(* IEC 61131-3 sources: std_i2980_v2.06_cp053/Source/IMM/ieccontrol/CentralCoordination1, 6 files *)

(* ---- ABActiveMovements.pu ---- *)
(*
@h    ! WARNING !
@h    The Kemro K2 system (including software) only meets category B according to EN 954-1,
@h    thus it is not intended for usage in safety-relevant control applications in the field
@h    of personal safety (e.g. emergency stop).
@h    To implement potentially necessary safety-relevant control tasks, always use additional
@h    external safety devices that are intended for the particular purpose, and meet the necessary
@h    functional safety.
@h    For further information see EN 954-1 (EN ISO 13849-1) and/or the K2-x00 user manual, chapter
@h    "CE conformity, directives and standards".

*)

IMPORT_OVER_LISTFILE
 SET_ALARM
, cCompNone
, cMoveNone
, cCompInjection
, cMinMoveIdent
, cMaxActiveMovements
, cMoveFwd
, tevMovementState
, tyMovementRegisterList
, tsActiveMovements
, tsStartedMoveData
, tyNumberOfDevices
, tyInjectHoldNumbers
, tevStartedStopped
, tevMovementStateData
, FBGetMoveNumber
, tevStartedStoppedData

END_IMPORT

ALGORITHM_BLOCK ABActiveMovements #DUMMY_EDIT_BLOCK

SYSTEM_VAR
 sv_MovementsAvailable : tyMovementRegisterList;
 sv_iMovementsAvailable : DINT;
 sv_ActiveMovements : tsActiveMovements;
 sv_StartedMovements : tsStartedMoveData;
 sv_bInitDone : BOOL;
 sv_NumberOfDevices : tyNumberOfDevices;
END_VAR

SYSTEM_OBJECT
 EV_Task_3 : TASK;
 evMovementState : tevMovementState;
 PU_Task_13 : TASK;
 evStartedStopped : tevStartedStopped;
 erMaxStartedMovementsExceeded : ALARM;
 erMaxActiveMovementsExceeded : ALARM;
END_OBJECT

VAR
 InjectHoldNumbers : tyInjectHoldNumbers;
END_VAR

(*
Manage a list of active movements for displaying
the active movement on the HMI.
Reacts to evMovementState events
*)

EVENT_ALGORITHM evaMovementState ON EV_Task_3 WITH evMovementState

VAR_INPUT
 evMovementStateData : tevMovementStateData;
END_VAR

VAR_TEMP
 i : DINT;
 k : DINT;
END_VAR

VAR
 iMoveNumber : DINT;
 MovementStateData : tevMovementStateData;
 fbGetMoveNumber : FBGetMoveNumber;
END_VAR
#BEGIN_EDIT_BLOCK
(**************************************** WARNING ********************************************
 *** The KEBA Kemro K2 System including software is not intended for safety control tasks! ***
 ***                       For further information see Comment tab!                        ***
 *********************************************************************************************)

MovementStateData := evMovementStateData;

IF MovementStateData.State = nInactive AND MovementStateData.DeviceId.CompId = cCompInjection AND
   MovementStateData.MoveDir = cMoveFwd AND MovementStateData.MoveId = cMoveInject THEN
   //inject movement was stopped -> check if holding was active
    IF InjectHoldNumbers[MovementStateData.DeviceId.IndexId].bHoldActive THEN
        //holding was active
        iMoveNumber := InjectHoldNumbers[MovementStateData.DeviceId.IndexId].iHoldMovement;
    ELSE
        //holding was not active
        iMoveNumber := InjectHoldNumbers[MovementStateData.DeviceId.IndexId].iInjectMovement;
    END_IF;
    InjectHoldNumbers[MovementStateData.DeviceId.IndexId].bHoldActive := FALSE;
ELSE
    // -> get movement number
    fbGetMoveNumber(DeviceId := MovementStateData.DeviceId,
                    MoveId := MovementStateData.MoveId,
                    MoveDir := MovementStateData.MoveDir,
                    iMoveNumber => iMoveNumber);
END_IF;

IF (iMoveNumber = 0) THEN
    //no movement found
    RETURN;
END_IF;

IF MovementStateData.State = nActive THEN
    IF MovementStateData.MoveId = cMoveHold THEN
        // hold phase active -> search inject movement and change number to hold movement
        FOR i := 1 TO sv_ActiveMovements.iNumberOfActiveMovements DO
            IF sv_ActiveMovements.ActiveMovements[i] = InjectHoldNumbers[MovementStateData.DeviceId.IndexId].iInjectMovement THEN
                sv_ActiveMovements.ActiveMovements[i] := InjectHoldNumbers[MovementStateData.DeviceId.IndexId].iHoldMovement;
                InjectHoldNumbers[MovementStateData.DeviceId.IndexId].bHoldActive := TRUE;
                EXIT;
            END_IF;
        END_FOR;
    ELSE
        IF sv_ActiveMovements.iNumberOfActiveMovements < cMaxActiveMovements THEN
            //movement was started -> add movement to list
            sv_ActiveMovements.ActiveMovements[(sv_ActiveMovements.iNumberOfActiveMovements+1)] := iMoveNumber;
            sv_ActiveMovements.iNumberOfActiveMovements := sv_ActiveMovements.iNumberOfActiveMovements + 1;
        ELSE
            //too many movements active
            SET_ALARM(Name := erMaxActiveMovementsExceeded,
                      SubID1 := cMaxActiveMovements);
        END_IF;
    END_IF;
ELSE
    //movement was stopped -> find movement and delete it from array
    FOR i := 1 TO sv_ActiveMovements.iNumberOfActiveMovements DO
        IF sv_ActiveMovements.ActiveMovements[i] = iMoveNumber THEN
            sv_ActiveMovements.ActiveMovements[i] := 0;
            //move all other movements so that there is no empty field in the list
            FOR k:= (i+1) TO cMaxActiveMovements DO
                sv_ActiveMovements.ActiveMovements[(k-1)] := sv_ActiveMovements.ActiveMovements[k];
                sv_ActiveMovements.ActiveMovements[k] := 0;
            END_FOR;
            sv_ActiveMovements.iNumberOfActiveMovements := sv_ActiveMovements.iNumberOfActiveMovements -1;
            EXIT;
        END_IF;
    END_FOR;

END_IF;

;#END_EDIT_BLOCK END_ALGORITHM

(*
Manage list and count of currently started movments
in sv_StartedMovements when receiving evStartedStopped events
*)

EVENT_ALGORITHM evaStartedStopped ON EV_Task_3 WITH evStartedStopped

VAR_INPUT
 evStartedStoppedData : tevStartedStoppedData;
END_VAR

VAR_TEMP
 i : DINT;
END_VAR

VAR
 dummy : DINT;
END_VAR
#BEGIN_EDIT_BLOCK
(**************************************** WARNING ********************************************
 *** The KEBA Kemro K2 System including software is not intended for safety control tasks! ***
 ***                       For further information see Comment tab!                        ***
 *********************************************************************************************)

IF evStartedStoppedData.State = nStarted THEN
    //movement started
    IF sv_StartedMovements.iStartedMovements < cMaxActiveMovements THEN
        //add movement to sv_StartedMovements
        sv_StartedMovements.iStartedMovements := sv_StartedMovements.iStartedMovements +1;
        sv_StartedMovements.MoveData[sv_StartedMovements.iStartedMovements].DeviceId := evStartedStoppedData.DeviceId;
        sv_StartedMovements.MoveData[sv_StartedMovements.iStartedMovements].MoveDir := evStartedStoppedData.MoveDir;
        sv_StartedMovements.MoveData[sv_StartedMovements.iStartedMovements].MoveId := evStartedStoppedData.MoveId;
    ELSE
        //too many movements started
        //show some information about the movement to make debugging easier
        dummy := Print('set alarm erMaxStartedMovementsExceeded in ABActiveMovements.pu');
        dummy := Print('max. active movements: %d', cMaxActiveMovements);
        dummy := Print('tried to start    %d.%d %d/%d',
                       evStartedStoppedData.DeviceId.CompId, evStartedStoppedData.DeviceId.IndexId,
                       evStartedStoppedData.MoveId, evStartedStoppedData.MoveDir);
        FOR i := 1 TO cMaxActiveMovements DO
            dummy := Print('already started %d %d.%d %d/%d',
                           i, sv_StartedMovements.MoveData[i].DeviceId.CompId, sv_StartedMovements.MoveData[i].DeviceId.IndexId,
                           sv_StartedMovements.MoveData[i].MoveId, sv_StartedMovements.MoveData[i].MoveDir);
        END_FOR;

        //set alarm after tracing out
        SET_ALARM(Name := erMaxStartedMovementsExceeded,
                  SubID1 := cMaxActiveMovements);
    END_IF;
ELSE
    //movement stopped
    //remove movement from list with started movements
    FOR i := 1 TO sv_StartedMovements.iStartedMovements DO
        IF sv_StartedMovements.MoveData[i].DeviceId = evStartedStoppedData.DeviceId AND
           sv_StartedMovements.MoveData[i].MoveDir = evStartedStoppedData.MoveDir AND
           sv_StartedMovements.MoveData[i].MoveId = evStartedStoppedData.MoveId THEN
            sv_StartedMovements.MoveData[i].DeviceId.CompId := cCompNone;
            sv_StartedMovements.MoveData[i].DeviceId.IndexId := 1;
            sv_StartedMovements.MoveData[i].MoveDir := cMoveNone;
            sv_StartedMovements.MoveData[i].MoveId := cMinMoveIdent;
            //copy last entry in the list to this empty field
            sv_StartedMovements.MoveData[i] := sv_StartedMovements.MoveData[sv_StartedMovements.iStartedMovements];
            sv_StartedMovements.iStartedMovements := sv_StartedMovements.iStartedMovements -1;
            EXIT;
        END_IF;
    END_FOR;
END_IF;

;#END_EDIT_BLOCK END_ALGORITHM

POSTUPDATE_ALGORITHM pGetInjectHoldNumbers ON PU_Task_13 WITH sv_bInitDone

VAR_TEMP
 i : DINT;
 iDevice : DINT;
END_VAR
#BEGIN_EDIT_BLOCK
(**************************************** WARNING ********************************************
 *** The KEBA Kemro K2 System including software is not intended for safety control tasks! ***
 ***                       For further information see Comment tab!                        ***
 *********************************************************************************************)

//get icon pathes for inject and hold of all registered injection function units
FOR iDevice := 1 TO sv_NumberOfDevices[cCompInjection] DO

    FOR i := 1 TO sv_iMovementsAvailable DO
        IF sv_MovementsAvailable[i].DeviceId.CompId = cCompInjection AND
           sv_MovementsAvailable[i].pMovementData^.MoveId = cMoveInject THEN
            //save number of inject movement
            InjectHoldNumbers[sv_MovementsAvailable[i].DeviceId.IndexId].iInjectMovement := i;
        END_IF;
        IF sv_MovementsAvailable[i].DeviceId.CompId = cCompInjection AND
           sv_MovementsAvailable[i].pMovementData^.MoveId = cMoveHold THEN
            //save number of holding movement
            InjectHoldNumbers[sv_MovementsAvailable[i].DeviceId.IndexId].iHoldMovement := i;
        END_IF;
    END_FOR;

END_FOR;

;#END_EDIT_BLOCK END_ALGORITHM

END_ALGORITHM_BLOCK

#END_OF_IEC_PART

@Puma @IecEditor 6 86 @Pou 25
@@@BEG_Comment@@@
@h    ! WARNING !
@h    The Kemro K2 system (including software) only meets category B according to EN 954-1,
@h    thus it is not intended for usage in safety-relevant control applications in the field
@h    of personal safety (e.g. emergency stop).
@h    To implement potentially necessary safety-relevant control tasks, always use additional
@h    external safety devices that are intended for the particular purpose, and meet the necessary
@h    functional safety.
@h    For further information see EN 954-1 (EN ISO 13849-1) and/or the K2-x00 user manual, chapter
@h    "CE conformity, directives and standards".

@@@END_Comment@@@

@BEG_Contents

@BEG_Func
@RT(17)FuncTreeContainer
1
@Var @RT(9)SET_ALARM @RT(0) @T @T @DERIVED 0 @F @RT(23)KEBA_STANDARD_PROCEDURE @F
@T
@BEG_Attrib
0 @RT(0) @RT(0)
@END_Attrib
1 1 @F @F @F @F

@END_Func

@BEG_Const
@RT(18)ConstTreeContainer
6
@Var @RT(9)cCompNone @RT(0) @T @F @DT @RT(4)DINT @RT(0) @T @T @BASIC 0 @F
@F @F
@T
@BEG_Attrib
0 @RT(10)cMinCompId @RT(4)None
@END_Attrib
1 1 @F @F @F @F

@Var @RT(9)cMoveNone @RT(0) @T @F @DT @RT(4)DINT @RT(0) @T @T @BASIC 0 @F
@F @F
@T
@BEG_Attrib
0 @RT(13)cMinMoveIdent @RT(4)None
@END_Attrib
1 1 @F @F @F @F

@Var @RT(14)cCompInjection @RT(0) @T @F @DT @RT(4)DINT @RT(0) @T @T @BASIC 0 @F
@F @F
@T
@BEG_Attrib
0 @RT(3)104 @RT(19)Component Injection
@END_Attrib
1 1 @F @F @F @F

@Var @RT(13)cMinMoveIdent @RT(0) @T @F @DT @RT(4)DINT @RT(0) @T @T @BASIC 0 @F
@F @F
@T
@BEG_Attrib
0 @RT(1)1 @RT(32)lower limit for MoveId / MoveDir
@END_Attrib
1 1 @F @F @F @F

@Var @RT(19)cMaxActiveMovements @RT(0) @T @F @DT @RT(4)DINT @RT(0) @T @T @BASIC 0 @F
@F @F
@T
@BEG_Attrib
0 @RT(1)6 @RT(52)number of movements that are active at the same time
@END_Attrib
1 1 @F @F @F @F

@Var @RT(8)cMoveFwd @RT(0) @T @F @DT @RT(4)DINT @RT(0) @T @T @BASIC 0 @F
@F @F
@T
@BEG_Attrib
0 @RT(2)12 @RT(16)movement forward
@END_Attrib
1 1 @F @F @F @F

@END_Const

@BEG_Export

@BEG_Kind
@ALGORITHM_BLOCK @RT(17)ABActiveMovements @STRUCTURED_TEXT
@RT(0) @RT(0) @RT(0)
@END_Kind

@BEG_Dcl
@RT(16)DclTreeContainer
13
@Var @RT(9)EV_Task_3 @RT(0) @T @T @RENAMED 0 @T @T @DT @RT(4)TASK @RT(0) @T @T @BASIC 0 @F
@F @F
@T
@BEG_Attrib
3 @RT(0) @RT(0) @RT(0)
@END_Attrib
1 7 @F @F @F @F

@Var @RT(15)evMovementState @RT(0) @T @T @DERIVED 0 @T @T @DT @RT(16)tevMovementState @RT(0) @T @T @UNKNOWN 0 @F
@F @F
@T
@BEG_Attrib
3 @RT(0) @RT(0) @RT(0)
@END_Attrib
1 7 @F @F @F @F

@Var @RT(21)sv_MovementsAvailable @RT(0) @T @T @DERIVED 0 @T @T @DT @RT(22)tyMovementRegisterList @RT(0) @T @T @UNKNOWN 0 @F
@F @F
@T
@BEG_Attrib
3 @RT(0) @RT(0) @RT(0)
@END_Attrib
1 8 @F @F @F @F

@Var @RT(22)sv_iMovementsAvailable @RT(0) @T @F @DT @RT(4)DINT @RT(0) @T @T @BASIC 0 @F
@F @F
@T
@BEG_Attrib
3 @RT(0) @RT(0) @RT(0)
@END_Attrib
1 8 @F @F @F @F

@Var @RT(18)sv_ActiveMovements @RT(0) @T @T @DERIVED 0 @T @T @DT @RT(17)tsActiveMovements @RT(0) @T @T @UNKNOWN 0 @F
@F @F
@T
@BEG_Attrib
3 @RT(0) @RT(0) @RT(0)
@END_Attrib
1 8 @F @F @F @F

@Var @RT(19)sv_StartedMovements @RT(0) @T @T @DERIVED 0 @T @T @DT @RT(17)tsStartedMoveData @RT(0) @T @T @UNKNOWN 0 @F
@F @F
@T
@BEG_Attrib
3 @RT(0) @RT(0) @RT(0)
@END_Attrib
1 8 @F @F @F @F

@Var @RT(10)PU_Task_13 @RT(0) @T @T @RENAMED 0 @T @T @DT @RT(4)TASK @RT(0) @T @T @BASIC 0 @F
@F @F
@T
@BEG_Attrib
3 @RT(0) @RT(0) @RT(0)
@END_Attrib
1 7 @F @F @F @F

@Var @RT(12)sv_bInitDone @RT(0) @T @T @RENAMED 0 @T @T @DT @RT(4)BOOL @RT(0) @T @T @BASIC 0 @F
@F @F
@T
@BEG_Attrib
3 @RT(0) @RT(0) @RT(0)
@END_Attrib
1 8 @F @F @F @F

@Var @RT(18)sv_NumberOfDevices @RT(0) @T @T @DERIVED 0 @T @T @DT @RT(17)tyNumberOfDevices @RT(0) @T @T @UNKNOWN 0 @F
@F @F
@T
@BEG_Attrib
3 @RT(0) @RT(0) @RT(0)
@END_Attrib
1 8 @F @F @F @F

@Var @RT(17)InjectHoldNumbers @RT(0) @T @T @DERIVED 0 @T @T @DT @RT(19)tyInjectHoldNumbers @RT(0) @T @T @UNKNOWN 0 @F
@F @F
@T
@BEG_Attrib
3 @RT(0) @RT(0) @RT(0)
@END_Attrib
1 0 @F @F @F @F

@Var @RT(16)evStartedStopped @RT(0) @T @T @RENAMED 0 @T @T @DT @RT(17)tevStartedStopped @RT(0) @T @T @UNKNOWN 0 @F
@F @F
@T
@BEG_Attrib
3 @RT(0) @RT(0) @RT(0)
@END_Attrib
1 7 @F @F @F @F

@Var @RT(29)erMaxStartedMovementsExceeded @RT(0) @T @T @RENAMED 0 @T @T @DT @RT(5)ALARM @RT(0) @T @T @BASIC 0 @F
@F @F
@T
@BEG_Attrib
3 @RT(0) @RT(0) @RT(0)
@END_Attrib
1 7 @F @F @F @F

@Var @RT(28)erMaxActiveMovementsExceeded @RT(0) @T @T @RENAMED 0 @T @T @DT @RT(5)ALARM @RT(0) @T @T @BASIC 0 @F
@F @F
@T
@BEG_Attrib
3 @RT(0) @RT(0) @RT(0)
@END_Attrib
1 7 @F @F @F @F

@END_Dcl

@END_Export

@BEG_Body

3

@BEG_Export

@BEG_Algo
@EVENT_ALGORITHM @RT(16)evaMovementState @STRUCTURED_TEXT
@RT(0) @RT(15)evMovementState @RT(9)EV_Task_3 @F @F
@END_Algo

@BEG_Dcl
@RT(16)DclTreeContainer
6
@Var @RT(19)evMovementStateData @RT(0) @T @T @DERIVED 0 @T @T @DT @RT(20)tevMovementStateData @RT(0) @T @T @UNKNOWN 0 @F
@F @F
@T
@BEG_Attrib
3 @RT(0) @RT(0) @RT(0)
@END_Attrib
1 1 @F @F @F @F

@Var @RT(1)i @RT(0) @T @F @DT @RT(4)DINT @RT(0) @T @T @BASIC 0 @F
@F @F
@T
@BEG_Attrib
3 @RT(0) @RT(0) @RT(0)
@END_Attrib
1 4 @F @F @F @F

@Var @RT(1)k @RT(0) @T @F @DT @RT(4)DINT @RT(0) @T @T @BASIC 0 @F
@F @F
@T
@BEG_Attrib
3 @RT(0) @RT(0) @RT(0)
@END_Attrib
1 4 @F @F @F @F

@Var @RT(11)iMoveNumber @RT(0) @T @F @DT @RT(4)DINT @RT(0) @T @T @BASIC 0 @F
@F @F
@T
@BEG_Attrib
3 @RT(0) @RT(0) @RT(0)
@END_Attrib
1 0 @F @F @F @F

@Var @RT(17)MovementStateData @RT(0) @T @T @DERIVED 0 @T @T @DT @RT(20)tevMovementStateData @RT(0) @T @T @UNKNOWN 0 @F
@F @F
@T
@BEG_Attrib
3 @RT(0) @RT(0) @RT(0)
@END_Attrib
1 0 @F @F @F @F

@Var @RT(15)fbGetMoveNumber @RT(0) @T @T @DERIVED 0 @T @T @DT @RT(15)FBGetMoveNumber @RT(0) @T @T @UNKNOWN 0 @F
@F @F
@T
@BEG_Attrib
3 @RT(0) @RT(0) @RT(0)
@END_Attrib
1 0 @F @F @F @F

@END_Dcl

@END_Export

@BEG_Export

@BEG_Algo
@EVENT_ALGORITHM @RT(17)evaStartedStopped @STRUCTURED_TEXT
@RT(0) @RT(16)evStartedStopped @RT(9)EV_Task_3 @F @F
@END_Algo

@BEG_Dcl
@RT(16)DclTreeContainer
3
@Var @RT(20)evStartedStoppedData @RT(0) @T @T @DERIVED 0 @T @T @DT @RT(21)tevStartedStoppedData @RT(0) @T @T @UNKNOWN 0 @F
@F @F
@T
@BEG_Attrib
3 @RT(0) @RT(0) @RT(0)
@END_Attrib
1 1 @F @F @F @F

@Var @RT(1)i @RT(0) @T @F @DT @RT(4)DINT @RT(0) @T @T @BASIC 0 @F
@F @F
@T
@BEG_Attrib
3 @RT(0) @RT(0) @RT(0)
@END_Attrib
1 4 @F @F @F @F

@Var @RT(5)dummy @RT(0) @T @F @DT @RT(4)DINT @RT(0) @T @T @BASIC 0 @F
@F @F
@T
@BEG_Attrib
3 @RT(0) @RT(0) @RT(0)
@END_Attrib
1 0 @F @F @F @F

@END_Dcl

@END_Export

@BEG_Export

@BEG_Algo
@POSTUPDATE_ALGORITHM @RT(21)pGetInjectHoldNumbers @STRUCTURED_TEXT
@RT(0) @RT(12)sv_bInitDone @RT(10)PU_Task_13 @F @F
@END_Algo

@BEG_Dcl
@RT(16)DclTreeContainer
2
@Var @RT(1)i @RT(0) @T @F @DT @RT(4)DINT @RT(0) @T @T @BASIC 0 @F
@F @F
@T
@BEG_Attrib
3 @RT(0) @RT(0) @RT(0)
@END_Attrib
1 4 @F @F @F @F

@Var @RT(7)iDevice @RT(0) @T @F @DT @RT(4)DINT @RT(0) @T @T @BASIC 0 @F
@F @F
@T
@BEG_Attrib
3 @RT(0) @RT(0) @RT(0)
@END_Attrib
1 4 @F @F @F @F

@END_Dcl

@END_Export

@BEG_Body
@TL(72)
(**************************************** WARNING ********************************************
 *** The KEBA Kemro K2 System including software is not intended for safety control tasks! ***
 ***                       For further information see Comment tab!                        ***
 *********************************************************************************************)

MovementStateData := evMovementStateData;

IF MovementStateData.State = nInactive AND MovementStateData.DeviceId.CompId = cCompInjection AND
   MovementStateData.MoveDir = cMoveFwd AND MovementStateData.MoveId = cMoveInject THEN
   //inject movement was stopped -> check if holding was active
    IF InjectHoldNumbers[MovementStateData.DeviceId.IndexId].bHoldActive THEN
        //holding was active
        iMoveNumber := InjectHoldNumbers[MovementStateData.DeviceId.IndexId].iHoldMovement;
    ELSE
        //holding was not active
        iMoveNumber := InjectHoldNumbers[MovementStateData.DeviceId.IndexId].iInjectMovement;
    END_IF;
    InjectHoldNumbers[MovementStateData.DeviceId.IndexId].bHoldActive := FALSE;
ELSE
    // -> get movement number
    fbGetMoveNumber(DeviceId := MovementStateData.DeviceId,
                    MoveId := MovementStateData.MoveId,
                    MoveDir := MovementStateData.MoveDir,
                    iMoveNumber => iMoveNumber);
END_IF;

IF (iMoveNumber = 0) THEN
    //no movement found
    RETURN;
END_IF;

IF MovementStateData.State = nActive THEN
    IF MovementStateData.MoveId = cMoveHold THEN
        // hold phase active -> search inject movement and change number to hold movement
        FOR i := 1 TO sv_ActiveMovements.iNumberOfActiveMovements DO
            IF sv_ActiveMovements.ActiveMovements[i] = InjectHoldNumbers[MovementStateData.DeviceId.IndexId].iInjectMovement THEN
                sv_ActiveMovements.ActiveMovements[i] := InjectHoldNumbers[MovementStateData.DeviceId.IndexId].iHoldMovement;
                InjectHoldNumbers[MovementStateData.DeviceId.IndexId].bHoldActive := TRUE;
                EXIT;
            END_IF;
        END_FOR;
    ELSE
        IF sv_ActiveMovements.iNumberOfActiveMovements < cMaxActiveMovements THEN
            //movement was started -> add movement to list
            sv_ActiveMovements.ActiveMovements[(sv_ActiveMovements.iNumberOfActiveMovements+1)] := iMoveNumber;
            sv_ActiveMovements.iNumberOfActiveMovements := sv_ActiveMovements.iNumberOfActiveMovements + 1;
        ELSE
            //too many movements active
            SET_ALARM(Name := erMaxActiveMovementsExceeded,
                      SubID1 := cMaxActiveMovements);
        END_IF;
    END_IF;
ELSE
    //movement was stopped -> find movement and delete it from array
    FOR i := 1 TO sv_ActiveMovements.iNumberOfActiveMovements DO
        IF sv_ActiveMovements.ActiveMovements[i] = iMoveNumber THEN
            sv_ActiveMovements.ActiveMovements[i] := 0;
            //move all other movements so that there is no empty field in the list
            FOR k:= (i+1) TO cMaxActiveMovements DO
                sv_ActiveMovements.ActiveMovements[(k-1)] := sv_ActiveMovements.ActiveMovements[k];
                sv_ActiveMovements.ActiveMovements[k] := 0;
            END_FOR;
            sv_ActiveMovements.iNumberOfActiveMovements := sv_ActiveMovements.iNumberOfActiveMovements -1;
            EXIT;
        END_IF;
    END_FOR;

END_IF;

@END_Body

@@@BEG_Comment@@@
@TL(3)
Manage a list of active movements for displaying
the active movement on the HMI.
Reacts to evMovementState events
@@@END_Comment@@@

@BEG_Body
@TL(54)
(**************************************** WARNING ********************************************
 *** The KEBA Kemro K2 System including software is not intended for safety control tasks! ***
 ***                       For further information see Comment tab!                        ***
 *********************************************************************************************)

IF evStartedStoppedData.State = nStarted THEN
    //movement started
    IF sv_StartedMovements.iStartedMovements < cMaxActiveMovements THEN
        //add movement to sv_StartedMovements
        sv_StartedMovements.iStartedMovements := sv_StartedMovements.iStartedMovements +1;
        sv_StartedMovements.MoveData[sv_StartedMovements.iStartedMovements].DeviceId := evStartedStoppedData.DeviceId;
        sv_StartedMovements.MoveData[sv_StartedMovements.iStartedMovements].MoveDir := evStartedStoppedData.MoveDir;
        sv_StartedMovements.MoveData[sv_StartedMovements.iStartedMovements].MoveId := evStartedStoppedData.MoveId;
    ELSE
        //too many movements started
        //show some information about the movement to make debugging easier
        dummy := Print('set alarm erMaxStartedMovementsExceeded in ABActiveMovements.pu');
        dummy := Print('max. active movements: %d', cMaxActiveMovements);
        dummy := Print('tried to start    %d.%d %d/%d',
                       evStartedStoppedData.DeviceId.CompId, evStartedStoppedData.DeviceId.IndexId,
                       evStartedStoppedData.MoveId, evStartedStoppedData.MoveDir);
        FOR i := 1 TO cMaxActiveMovements DO
            dummy := Print('already started %d %d.%d %d/%d',
                           i, sv_StartedMovements.MoveData[i].DeviceId.CompId, sv_StartedMovements.MoveData[i].DeviceId.IndexId,
                           sv_StartedMovements.MoveData[i].MoveId, sv_StartedMovements.MoveData[i].MoveDir);
        END_FOR;

        //set alarm after tracing out
        SET_ALARM(Name := erMaxStartedMovementsExceeded,
                  SubID1 := cMaxActiveMovements);
    END_IF;
ELSE
    //movement stopped
    //remove movement from list with started movements
    FOR i := 1 TO sv_StartedMovements.iStartedMovements DO
        IF sv_StartedMovements.MoveData[i].DeviceId = evStartedStoppedData.DeviceId AND
           sv_StartedMovements.MoveData[i].MoveDir = evStartedStoppedData.MoveDir AND
           sv_StartedMovements.MoveData[i].MoveId = evStartedStoppedData.MoveId THEN
            sv_StartedMovements.MoveData[i].DeviceId.CompId := cCompNone;
            sv_StartedMovements.MoveData[i].DeviceId.IndexId := 1;
            sv_StartedMovements.MoveData[i].MoveDir := cMoveNone;
            sv_StartedMovements.MoveData[i].MoveId := cMinMoveIdent;
            //copy last entry in the list to this empty field
            sv_StartedMovements.MoveData[i] := sv_StartedMovements.MoveData[sv_StartedMovements.iStartedMovements];
            sv_StartedMovements.iStartedMovements := sv_StartedMovements.iStartedMovements -1;
            EXIT;
        END_IF;
    END_FOR;
END_IF;

@END_Body

@@@BEG_Comment@@@
@TL(2)
Manage list and count of currently started movments
in sv_StartedMovements when receiving evStartedStopped events
@@@END_Comment@@@

@BEG_Body
@TL(23)
(**************************************** WARNING ********************************************
 *** The KEBA Kemro K2 System including software is not intended for safety control tasks! ***
 ***                       For further information see Comment tab!                        ***
 *********************************************************************************************)

//get icon pathes for inject and hold of all registered injection function units
FOR iDevice := 1 TO sv_NumberOfDevices[cCompInjection] DO

    FOR i := 1 TO sv_iMovementsAvailable DO
        IF sv_MovementsAvailable[i].DeviceId.CompId = cCompInjection AND
           sv_MovementsAvailable[i].pMovementData^.MoveId = cMoveInject THEN
            //save number of inject movement
            InjectHoldNumbers[sv_MovementsAvailable[i].DeviceId.IndexId].iInjectMovement := i;
        END_IF;
        IF sv_MovementsAvailable[i].DeviceId.CompId = cCompInjection AND
           sv_MovementsAvailable[i].pMovementData^.MoveId = cMoveHold THEN
            //save number of holding movement
            InjectHoldNumbers[sv_MovementsAvailable[i].DeviceId.IndexId].iHoldMovement := i;
        END_IF;
    END_FOR;

END_FOR;

@END_Body

@@@BEG_Comment@@@
@TL(0)

@@@END_Comment@@@
@END_Body

@END_Contents
@@@BEG_Password@@@
M2hzZmhrMw==
@@@END_Password@@@

(* ---- ABAvailableDevices.pu ---- *)
(*
@h    ! WARNING !
@h    The Kemro K2 system (including software) only meets category B according to EN 954-1,
@h    thus it is not intended for usage in safety-relevant control applications in the field
@h    of personal safety (e.g. emergency stop).
@h    To implement potentially necessary safety-relevant control tasks, always use additional
@h    external safety devices that are intended for the particular purpose, and meet the necessary
@h    functional safety.
@h    For further information see EN 954-1 (EN ISO 13849-1) and/or the K2-x00 user manual, chapter
@h    "CE conformity, directives and standards".

This AB listens to the device register events and sets
the sv_CoreData[X].bAvailable - flag if a core is available (registered).
Additionally it listens to evCoreTypeChanged events and sets
sv_bCoresActive if any registered core is switched on.
After a failed creation of a new sequence (by using program switches), The core priorities are
checked. If there are some equal priorities, an according alarm is displayed
*)

IMPORT_OVER_LISTFILE
 SET_ALARM
, cCompAirValve
, cMaxDeviceIndex
, cMoveIn
, tyCoreData
, tevDeviceRegister
, tevCoreTypeChanged
, tyDeviceAvailable
, tyNumberOfDevices
, KSYS_Status
, tevDeviceRegisterData
, tevCoreTypeChangedData

END_IMPORT

ALGORITHM_BLOCK ABAvailableDevices #DUMMY_EDIT_BLOCK

SYSTEM_VAR
 sv_CoreData : tyCoreData;
 sv_CoreOff : tyDeviceAvailable;
 sv_bCoresActive : BOOL (* TRUE: any core is switched on *);
 sv_bInitStart : BOOL;
 sv_bUseProgramSwitches : BOOL;
 sv_bCoresParallelToMold : BOOL;
 sv_bDeviceRegisterDone : BOOL;
 sv_NumberOfDevices : tyNumberOfDevices;
END_VAR

SYSTEM_OBJECT
 EV_Task_3 : TASK;
 evDeviceRegister : tevDeviceRegister;
 EV_Task_7 : TASK;
 evCoreTypeChanged : tevCoreTypeChanged;
 PU_Task_7 : TASK;
 TaskMid : TASK;
 erEqualCorePriority : ALARM;
 PU_Task_3 : TASK;
END_OBJECT

VAR
 mpiODCSequenceUpdated : REFTO DINT;
 mpiODCInitOk : REFTO DINT;
END_VAR

POSTUPDATE_ALGORITHM pInitStart ON PU_Task_7 WITH sv_bInitStart

VAR
 state : KSYS_Status;
END_VAR
#BEGIN_EDIT_BLOCK
(**************************************** WARNING ********************************************
 *** The KEBA Kemro K2 System including software is not intended for safety control tasks! ***
 ***                       For further information see Comment tab!                        ***
 *********************************************************************************************)

//get references
mpiODCSequenceUpdated := GET_SYNC_REFTO('ODC1.sv_iODCSequenceUpdated', T#0s, state);
mpiODCInitOk := GET_SYNC_REFTO('ODC1.sv_iInitOK', T#0s, state);

;#END_EDIT_BLOCK END_ALGORITHM

(*
listen to register events of cores and airvalves and set according available flags
if a register event from a core or airvalve is received
*)

EVENT_ALGORITHM evaDeviceRegister ON EV_Task_3 WITH evDeviceRegister

VAR_INPUT
 evDeviceRegisterData : tevDeviceRegisterData;
END_VAR

VAR_TEMP
 i : DINT;
END_VAR

VAR
 bInitDone : BOOL;
END_VAR
#BEGIN_EDIT_BLOCK
(**************************************** WARNING ********************************************
 *** The KEBA Kemro K2 System including software is not intended for safety control tasks! ***
 ***                       For further information see Comment tab!                        ***
 *********************************************************************************************)

IF NOT bInitDone THEN
    //reset available flag for all possible cores because the whole structure sv_CoreData is retain!
    FOR i := 1 TO cMaxDeviceIndex DO
        sv_CoreData[i].bAvailable := FALSE;
    END_FOR;
    bInitDone := TRUE;
END_IF;

CASE evDeviceRegisterData.DeviceId.CompId OF
   cCompCore:
      //set available flag of according Core FU
      sv_CoreData[evDeviceRegisterData.DeviceId.IndexId].bAvailable := TRUE;

END_CASE;

;#END_EDIT_BLOCK END_ALGORITHM

EVENT_ALGORITHM evaCoreTypeChanged ON EV_Task_7 WITH evCoreTypeChanged

VAR_INPUT
 evCoreTypeChangedData : tevCoreTypeChangedData;
END_VAR

VAR_TEMP
 i : DINT;
END_VAR
#BEGIN_EDIT_BLOCK
(**************************************** WARNING ********************************************
 *** The KEBA Kemro K2 System including software is not intended for safety control tasks! ***
 ***                       For further information see Comment tab!                        ***
 *********************************************************************************************)

sv_CoreOff[evCoreTypeChangedData.DeviceId.IndexId] := evCoreTypeChangedData.bCoreOff;

sv_bCoresActive := FALSE;
FOR i := 1 TO cMaxDeviceIndex DO
   IF sv_CoreData[i].bAvailable AND NOT sv_CoreOff[i] THEN
      //Core is available and not switched off
      sv_bCoresActive := TRUE;
   END_IF;
END_FOR;

;#END_EDIT_BLOCK END_ALGORITHM

POSTUPDATE_ALGORITHM pNewSequence ON PU_Task_7 WITH mpiODCSequenceUpdated^

#BEGIN_EDIT_BLOCK
(**************************************** WARNING ********************************************
 *** The KEBA Kemro K2 System including software is not intended for safety control tasks! ***
 ***                       For further information see Comment tab!                        ***
 *********************************************************************************************)

//new sequence created by using program switches -> check if creation was successful
//if not: check core priorities
IF sv_bUseProgramSwitches AND mpiODCInitOk^ = 0 THEN
   //check for equal core priorities
   START_PROCESS_ALGORITHM(paCheckCorePriorities);
END_IF;

;#END_EDIT_BLOCK END_ALGORITHM

PROCESS_ALGORITHM paCheckCorePriorities ON TaskMid

VAR_TEMP
 i : DINT;
 k : DINT;
END_VAR

VAR
 bSetAlarm : BOOL;
END_VAR
#BEGIN_EDIT_BLOCK
(**************************************** WARNING ********************************************
 *** The KEBA Kemro K2 System including software is not intended for safety control tasks! ***
 ***                       For further information see Comment tab!                        ***
 *********************************************************************************************)

//check core priorites if some of them are equal

FOR i := 1 TO (cMaxDeviceIndex - 1)  DO
   IF sv_CoreData[i].bAvailable AND NOT sv_CoreOff[i] THEN
      //core i is available and activated

      //compare core priorities with all other cores
      FOR k := (i + 1) TO cMaxDeviceIndex DO
         IF sv_CoreData[k].bAvailable AND NOT sv_CoreOff[k] THEN
            //core k is available and activated
            //compare core in priority with core in priority of all other cores
            IF (sv_CoreData[i].InMode = sv_CoreData[k].InMode) THEN
               //same mode -> check priority

               bSetAlarm := FALSE;
               IF sv_CoreData[i].InMode = nDuringMoldClose THEN
                  //mode "during" -> also consider sv_bCoresParallelToMold and the according position
                  IF sv_bCoresParallelToMold THEN
                     IF (sv_CoreData[i].iCoreInPriority = sv_CoreData[k].iCoreInPriority) THEN
                        //cores parallel to mold and same priority -> alarm
                        bSetAlarm := TRUE;
                     END_IF;
                  ELSE
                     IF (sv_CoreData[i].rCoreInPosition = sv_CoreData[k].rCoreInPosition) AND
                        (sv_CoreData[i].iCoreInPriority = sv_CoreData[k].iCoreInPriority) THEN
                        //cores not parallel and priority and position equal -> alarm
                        bSetAlarm := TRUE;
                     END_IF;
                  END_IF;
               ELSE
                  //mode before or after
                  IF (sv_CoreData[i].iCoreInPriority = sv_CoreData[k].iCoreInPriority) THEN
                     //same priority -> alarm
                     bSetAlarm := TRUE;
                  END_IF;
               END_IF;

               IF bSetAlarm THEN
                  //same mode and same priority -> alarm
                     SET_ALARM(Name := erEqualCorePriority,
                               SubID1 := i,
                               SubID2 := cMoveIn,
                               SubID3 := k,
                               SubID4 := cMoveIn);
               END_IF;
            END_IF; //end_if core in priority

            //compare core out priority with core out priority of all other cores
            IF (sv_CoreData[i].OutMode = sv_CoreData[k].OutMode) THEN
               //same mode -> check priority

               bSetAlarm := FALSE;
               IF (sv_CoreData[i].OutMode = nDuringMoldOpen) THEN
                  //mode "during" -> also consider sv_bCoresParallelToMold and the according position
                  IF sv_bCoresParallelToMold THEN
                     IF (sv_CoreData[i].iCoreOutPriority = sv_CoreData[k].iCoreOutPriority) THEN
                        //cores parallel to mold and same priority -> alarm
                        bSetAlarm := TRUE;
                     END_IF;
                  ELSE
                     IF (sv_CoreData[i].rCoreOutPosition = sv_CoreData[k].rCoreOutPosition) AND
                        (sv_CoreData[i].iCoreOutPriority = sv_CoreData[k].iCoreOutPriority) THEN
                        //cores not parallel and priority and position equal -> alarm
                        bSetAlarm := TRUE;
                     END_IF;
                  END_IF;
               ELSE
                  //mode before or after
                  IF (sv_CoreData[i].iCoreOutPriority = sv_CoreData[k].iCoreOutPriority) THEN
                     //same priority -> alarm
                     bSetAlarm := TRUE;
                  END_IF;
               END_IF;

               IF bSetAlarm THEN
                  //same mode and same priority -> alarm
                     SET_ALARM(Name := erEqualCorePriority,
                               SubID1 := i,
                               SubID2 := cMoveOut,
                               SubID3 := k,
                               SubID4 := cMoveOut);
               END_IF;
            END_IF; //end_if core out priority

         END_IF; //end_if core k
      END_FOR;  //end_for core k
   END_IF; //end_if core i available and activated
END_FOR;

STOP_PROCESS_ALGORITHM();

;#END_EDIT_BLOCK END_ALGORITHM

POSTUPDATE_ALGORITHM pDeviceRegister ON PU_Task_3 WITH sv_bDeviceRegisterDone

VAR_TEMP
 i : DINT;
END_VAR
#BEGIN_EDIT_BLOCK
(**************************************** WARNING ********************************************
 *** The KEBA Kemro K2 System including software is not intended for safety control tasks! ***
 ***                       For further information see Comment tab!                        ***
 *********************************************************************************************)

//correct init value of core out priority (-1)
FOR i := 1 TO cMaxDeviceIndex DO
   IF sv_CoreData[i].bAvailable AND sv_CoreData[i].iCoreOutPriority = -1 THEN
      IF i = 1 THEN
         //first core gets highest number (= number of available cores)
         sv_CoreData[i].iCoreOutPriority := sv_NumberOfDevices[cCompCore];
      ELSE
         //other cores get lower number than the predecessor
         sv_CoreData[i].iCoreOutPriority := sv_CoreData[(i - 1)].iCoreOutPriority - 1;
      END_IF;
   END_IF;
END_FOR;

;#END_EDIT_BLOCK END_ALGORITHM

END_ALGORITHM_BLOCK

#END_OF_IEC_PART

@Puma @IecEditor 6 30 @Pou 25
@@@BEG_Comment@@@
@h    ! WARNING !
@h    The Kemro K2 system (including software) only meets category B according to EN 954-1,
@h    thus it is not intended for usage in safety-relevant control applications in the field
@h    of personal safety (e.g. emergency stop).
@h    To implement potentially necessary safety-relevant control tasks, always use additional
@h    external safety devices that are intended for the particular purpose, and meet the necessary
@h    functional safety.
@h    For further information see EN 954-1 (EN ISO 13849-1) and/or the K2-x00 user manual, chapter
@h    "CE conformity, directives and standards".

This AB listens to the device register events and sets
the sv_CoreData[X].bAvailable - flag if a core is available (registered).
Additionally it listens to evCoreTypeChanged events and sets
sv_bCoresActive if any registered core is switched on.
After a failed creation of a new sequence (by using program switches), The core priorities are
checked. If there are some equal priorities, an according alarm is displayed
@@@END_Comment@@@

@BEG_Contents

@BEG_Func
@RT(17)FuncTreeContainer
1
@Var @RT(9)SET_ALARM @RT(0) @T @T @DERIVED 0 @F @RT(23)KEBA_STANDARD_PROCEDURE @F
@T
@BEG_Attrib
0 @RT(0) @RT(0)
@END_Attrib
1 1 @F @F @F @F

@END_Func

@BEG_Const
@RT(18)ConstTreeContainer
3
@Var @RT(13)cCompAirValve @RT(0) @T @F @DT @RT(4)DINT @RT(0) @T @T @BASIC 0 @F
@F @F
@T
@BEG_Attrib
0 @RT(3)118 @RT(19)Component Air Valve
@END_Attrib
1 1 @F @F @F @F

@Var @RT(15)cMaxDeviceIndex @RT(0) @T @F @DT @RT(4)DINT @RT(0) @T @T @BASIC 0 @F
@F @F
@T
@BEG_Attrib
0 @RT(2)10 @RT(39)maximum number of devices per component
@END_Attrib
1 1 @F @F @F @F

@Var @RT(7)cMoveIn @RT(0) @T @F @DT @RT(4)DINT @RT(0) @T @T @BASIC 0 @F
@F @F
@T
@BEG_Attrib
0 @RT(2)21 @RT(26)move in (for example core)
@END_Attrib
1 1 @F @F @F @F

@END_Const

@BEG_Export

@BEG_Kind
@ALGORITHM_BLOCK @RT(18)ABAvailableDevices @STRUCTURED_TEXT
@RT(0) @RT(0) @RT(0)
@END_Kind

@BEG_Dcl
@RT(16)DclTreeContainer
18
@Var @RT(11)sv_CoreData @RT(0) @T @T @DERIVED 0 @F @RT(10)tyCoreData @F
@T
@BEG_Attrib
3 @RT(0) @RT(0) @RT(0)
@END_Attrib
1 8 @F @F @F @F

@Var @RT(9)EV_Task_3 @RT(0) @T @T @RENAMED 0 @T @T @DT @RT(4)TASK @RT(0) @T @T @BASIC 0 @F
@F @F
@T
@BEG_Attrib
3 @RT(0) @RT(0) @RT(0)
@END_Attrib
1 7 @F @F @F @F

@Var @RT(16)evDeviceRegister @RT(0) @T @T @RENAMED 0 @T @T @DT @RT(17)tevDeviceRegister @RT(0) @T @T @UNKNOWN 0 @F
@F @F
@T
@BEG_Attrib
3 @RT(0) @RT(0) @RT(0)
@END_Attrib
1 7 @F @F @F @F

@Var @RT(9)EV_Task_7 @RT(0) @T @T @RENAMED 0 @T @T @DT @RT(4)TASK @RT(0) @T @T @BASIC 0 @F
@F @F
@T
@BEG_Attrib
3 @RT(0) @RT(0) @RT(0)
@END_Attrib
1 7 @F @F @F @F

@Var @RT(17)evCoreTypeChanged @RT(0) @T @T @RENAMED 0 @T @T @DT @RT(18)tevCoreTypeChanged @RT(0) @T @T @UNKNOWN 0 @F
@F @F
@T
@BEG_Attrib
3 @RT(0) @RT(0) @RT(0)
@END_Attrib
1 7 @F @F @F @F

@Var @RT(10)sv_CoreOff @RT(0) @T @T @DERIVED 0 @T @T @DT @RT(17)tyDeviceAvailable @RT(0) @T @T @UNKNOWN 0 @F
@F @F
@T
@BEG_Attrib
3 @RT(0) @RT(0) @RT(0)
@END_Attrib
1 8 @F @F @F @F

@Var @RT(15)sv_bCoresActive @RT(0) @T @F @DT @RT(4)BOOL @RT(0) @T @T @BASIC 0 @F
@F @F
@T
@BEG_Attrib
3 @RT(0) @RT(29)TRUE: any core is switched on @RT(0)
@END_Attrib
1 8 @F @F @F @F

@Var @RT(21)mpiODCSequenceUpdated @RT(0) @T @T @REFTO 0 @T @DT @RT(4)DINT @RT(0) @T @T @BASIC 0 @F
@F @F
@T
@BEG_Attrib
3 @RT(0) @RT(0) @RT(0)
@END_Attrib
1 0 @F @F @F @F

@Var @RT(12)mpiODCInitOk @RT(0) @T @T @REFTO 0 @T @DT @RT(4)DINT @RT(0) @T @T @BASIC 0 @F
@F @F
@T
@BEG_Attrib
3 @RT(0) @RT(0) @RT(0)
@END_Attrib
1 0 @F @F @F @F

@Var @RT(9)PU_Task_7 @RT(0) @T @T @RENAMED 0 @T @T @DT @RT(4)TASK @RT(0) @T @T @BASIC 0 @F
@F @F
@T
@BEG_Attrib
3 @RT(0) @RT(0) @RT(0)
@END_Attrib
1 7 @F @F @F @F

@Var @RT(7)TaskMid @RT(0) @T @T @RENAMED 0 @T @T @DT @RT(4)TASK @RT(0) @T @T @BASIC 0 @F
@F @F
@T
@BEG_Attrib
3 @RT(0) @RT(0) @RT(0)
@END_Attrib
1 7 @F @F @F @F

@Var @RT(13)sv_bInitStart @RT(0) @T @F @DT @RT(4)BOOL @RT(0) @T @T @BASIC 0 @F
@F @F
@T
@BEG_Attrib
3 @RT(0) @RT(0) @RT(0)
@END_Attrib
1 8 @F @F @F @F

@Var @RT(19)erEqualCorePriority @RT(0) @T @F @DT @RT(5)ALARM @RT(0) @T @T @BASIC 0 @F
@F @F
@T
@BEG_Attrib
3 @RT(0) @RT(0) @RT(0)
@END_Attrib
1 7 @F @F @F @F

@Var @RT(22)sv_bUseProgramSwitches @RT(0) @T @F @DT @RT(4)BOOL @RT(0) @T @T @BASIC 0 @F
@F @F
@T
@BEG_Attrib
3 @RT(0) @RT(0) @RT(0)
@END_Attrib
1 8 @F @F @F @F

@Var @RT(23)sv_bCoresParallelToMold @RT(0) @T @F @DT @RT(4)BOOL @RT(0) @T @T @BASIC 0 @F
@F @F
@T
@BEG_Attrib
3 @RT(0) @RT(0) @RT(0)
@END_Attrib
1 8 @F @F @F @F

@Var @RT(9)PU_Task_3 @RT(0) @T @T @RENAMED 0 @T @T @DT @RT(4)TASK @RT(0) @T @T @BASIC 0 @F
@F @F
@T
@BEG_Attrib
3 @RT(0) @RT(0) @RT(0)
@END_Attrib
1 7 @F @F @F @F

@Var @RT(22)sv_bDeviceRegisterDone @RT(0) @T @T @RENAMED 0 @T @T @DT @RT(4)BOOL @RT(0) @T @T @BASIC 0 @F
@F @F
@T
@BEG_Attrib
3 @RT(0) @RT(0) @RT(0)
@END_Attrib
1 8 @F @F @F @F

@Var @RT(18)sv_NumberOfDevices @RT(0) @T @T @DERIVED 0 @F @RT(17)tyNumberOfDevices @F
@T
@BEG_Attrib
3 @RT(0) @RT(0) @RT(0)
@END_Attrib
1 8 @F @F @F @F

@END_Dcl

@END_Export

@BEG_Body

6

@BEG_Export

@BEG_Algo
@POSTUPDATE_ALGORITHM @RT(10)pInitStart @STRUCTURED_TEXT
@RT(0) @RT(13)sv_bInitStart @RT(9)PU_Task_7 @F @F
@END_Algo

@BEG_Dcl
@RT(16)DclTreeContainer
1
@Var @RT(5)state @RT(0) @T @T @DERIVED 0 @T @T @DT @RT(11)KSYS_Status @RT(0) @T @T @UNKNOWN 0 @F
@F @F
@T
@BEG_Attrib
3 @RT(0) @RT(0) @RT(0)
@END_Attrib
1 0 @F @F @F @F

@END_Dcl

@END_Export

@BEG_Export

@BEG_Algo
@EVENT_ALGORITHM @RT(17)evaDeviceRegister @STRUCTURED_TEXT
@RT(0) @RT(16)evDeviceRegister @RT(9)EV_Task_3 @F @F
@END_Algo

@BEG_Dcl
@RT(16)DclTreeContainer
3
@Var @RT(20)evDeviceRegisterData @RT(0) @T @T @DERIVED 0 @T @T @DT @RT(21)tevDeviceRegisterData @RT(0) @T @T @UNKNOWN 0 @F
@F @F
@T
@BEG_Attrib
3 @RT(0) @RT(0) @RT(0)
@END_Attrib
1 1 @F @F @F @F

@Var @RT(9)bInitDone @RT(0) @T @F @DT @RT(4)BOOL @RT(0) @T @T @BASIC 0 @F
@F @F
@T
@BEG_Attrib
3 @RT(0) @RT(0) @RT(0)
@END_Attrib
1 0 @F @F @F @F

@Var @RT(1)i @RT(0) @T @F @DT @RT(4)DINT @RT(0) @T @T @BASIC 0 @F
@F @F
@T
@BEG_Attrib
3 @RT(0) @RT(0) @RT(0)
@END_Attrib
1 4 @F @F @F @F

@END_Dcl

@END_Export

@BEG_Export

@BEG_Algo
@EVENT_ALGORITHM @RT(18)evaCoreTypeChanged @STRUCTURED_TEXT
@RT(0) @RT(17)evCoreTypeChanged @RT(9)EV_Task_7 @F @F
@END_Algo

@BEG_Dcl
@RT(16)DclTreeContainer
2
@Var @RT(21)evCoreTypeChangedData @RT(0) @T @T @DERIVED 0 @T @T @DT @RT(22)tevCoreTypeChangedData @RT(0) @T @T @UNKNOWN 0 @F
@F @F
@T
@BEG_Attrib
3 @RT(0) @RT(0) @RT(0)
@END_Attrib
1 1 @F @F @F @F

@Var @RT(1)i @RT(0) @T @F @DT @RT(4)DINT @RT(0) @T @T @BASIC 0 @F
@F @F
@T
@BEG_Attrib
3 @RT(0) @RT(0) @RT(0)
@END_Attrib
1 4 @F @F @F @F

@END_Dcl

@END_Export

@BEG_Export

@BEG_Algo
@POSTUPDATE_ALGORITHM @RT(12)pNewSequence @STRUCTURED_TEXT
@RT(0) @RT(22)mpiODCSequenceUpdated^ @RT(9)PU_Task_7 @F @F
@END_Algo

@BEG_Dcl
@RT(16)DclTreeContainer
0
@END_Dcl

@END_Export

@BEG_Export

@BEG_Algo
@PROCESS_ALGORITHM @RT(21)paCheckCorePriorities @STRUCTURED_TEXT
@RT(0) @RT(0) @RT(7)TaskMid @F @F
@END_Algo

@BEG_Dcl
@RT(16)DclTreeContainer
3
@Var @RT(1)i @RT(0) @T @F @DT @RT(4)DINT @RT(0) @T @T @BASIC 0 @F
@F @F
@T
@BEG_Attrib
3 @RT(0) @RT(0) @RT(0)
@END_Attrib
1 4 @F @F @F @F

@Var @RT(1)k @RT(0) @T @T @RENAMED 0 @T @T @DT @RT(4)DINT @RT(0) @T @T @BASIC 0 @F
@F @F
@T
@BEG_Attrib
3 @RT(0) @RT(0) @RT(0)
@END_Attrib
1 4 @F @F @F @F

@Var @RT(9)bSetAlarm @RT(0) @T @F @DT @RT(4)BOOL @RT(0) @T @T @BASIC 0 @F
@F @F
@T
@BEG_Attrib
3 @RT(0) @RT(0) @RT(0)
@END_Attrib
1 0 @F @F @F @F

@END_Dcl

@END_Export

@BEG_Export

@BEG_Algo
@POSTUPDATE_ALGORITHM @RT(15)pDeviceRegister @STRUCTURED_TEXT
@RT(0) @RT(22)sv_bDeviceRegisterDone @RT(9)PU_Task_3 @F @F
@END_Algo

@BEG_Dcl
@RT(16)DclTreeContainer
1
@Var @RT(1)i @RT(0) @T @F @DT @RT(4)DINT @RT(0) @T @T @BASIC 0 @F
@F @F
@T
@BEG_Attrib
3 @RT(0) @RT(0) @RT(0)
@END_Attrib
1 4 @F @F @F @F

@END_Dcl

@END_Export

@BEG_Body
@TL(10)
(**************************************** WARNING ********************************************
 *** The KEBA Kemro K2 System including software is not intended for safety control tasks! ***
 ***                       For further information see Comment tab!                        ***
 *********************************************************************************************)

//get references
mpiODCSequenceUpdated := GET_SYNC_REFTO('ODC1.sv_iODCSequenceUpdated', T#0s, state);
mpiODCInitOk := GET_SYNC_REFTO('ODC1.sv_iInitOK', T#0s, state);

@END_Body

@@@BEG_Comment@@@
@TL(0)

@@@END_Comment@@@

@BEG_Body
@TL(20)
(**************************************** WARNING ********************************************
 *** The KEBA Kemro K2 System including software is not intended for safety control tasks! ***
 ***                       For further information see Comment tab!                        ***
 *********************************************************************************************)

IF NOT bInitDone THEN
    //reset available flag for all possible cores because the whole structure sv_CoreData is retain!
    FOR i := 1 TO cMaxDeviceIndex DO
        sv_CoreData[i].bAvailable := FALSE;
    END_FOR;
    bInitDone := TRUE;
END_IF;

CASE evDeviceRegisterData.DeviceId.CompId OF
   cCompCore:
      //set available flag of according Core FU
      sv_CoreData[evDeviceRegisterData.DeviceId.IndexId].bAvailable := TRUE;

END_CASE;

@END_Body

@@@BEG_Comment@@@
@TL(2)
listen to register events of cores and airvalves and set according available flags
if a register event from a core or airvalve is received
@@@END_Comment@@@

@BEG_Body
@TL(15)
(**************************************** WARNING ********************************************
 *** The KEBA Kemro K2 System including software is not intended for safety control tasks! ***
 ***                       For further information see Comment tab!                        ***
 *********************************************************************************************)

sv_CoreOff[evCoreTypeChangedData.DeviceId.IndexId] := evCoreTypeChangedData.bCoreOff;

sv_bCoresActive := FALSE;
FOR i := 1 TO cMaxDeviceIndex DO
   IF sv_CoreData[i].bAvailable AND NOT sv_CoreOff[i] THEN
      //Core is available and not switched off
      sv_bCoresActive := TRUE;
   END_IF;
END_FOR;

@END_Body

@@@BEG_Comment@@@
@TL(0)

@@@END_Comment@@@

@BEG_Body
@TL(12)
(**************************************** WARNING ********************************************
 *** The KEBA Kemro K2 System including software is not intended for safety control tasks! ***
 ***                       For further information see Comment tab!                        ***
 *********************************************************************************************)

//new sequence created by using program switches -> check if creation was successful
//if not: check core priorities
IF sv_bUseProgramSwitches AND mpiODCInitOk^ = 0 THEN
   //check for equal core priorities
   START_PROCESS_ALGORITHM(paCheckCorePriorities);
END_IF;

@END_Body

@@@BEG_Comment@@@
@TL(0)

@@@END_Comment@@@

@BEG_Body
@TL(97)
(**************************************** WARNING ********************************************
 *** The KEBA Kemro K2 System including software is not intended for safety control tasks! ***
 ***                       For further information see Comment tab!                        ***
 *********************************************************************************************)

//check core priorites if some of them are equal

FOR i := 1 TO (cMaxDeviceIndex - 1)  DO
   IF sv_CoreData[i].bAvailable AND NOT sv_CoreOff[i] THEN
      //core i is available and activated

      //compare core priorities with all other cores
      FOR k := (i + 1) TO cMaxDeviceIndex DO
         IF sv_CoreData[k].bAvailable AND NOT sv_CoreOff[k] THEN
            //core k is available and activated
            //compare core in priority with core in priority of all other cores
            IF (sv_CoreData[i].InMode = sv_CoreData[k].InMode) THEN
               //same mode -> check priority

               bSetAlarm := FALSE;
               IF sv_CoreData[i].InMode = nDuringMoldClose THEN
                  //mode "during" -> also consider sv_bCoresParallelToMold and the according position
                  IF sv_bCoresParallelToMold THEN
                     IF (sv_CoreData[i].iCoreInPriority = sv_CoreData[k].iCoreInPriority) THEN
                        //cores parallel to mold and same priority -> alarm
                        bSetAlarm := TRUE;
                     END_IF;
                  ELSE
                     IF (sv_CoreData[i].rCoreInPosition = sv_CoreData[k].rCoreInPosition) AND
                        (sv_CoreData[i].iCoreInPriority = sv_CoreData[k].iCoreInPriority) THEN
                        //cores not parallel and priority and position equal -> alarm
                        bSetAlarm := TRUE;
                     END_IF;
                  END_IF;
               ELSE
                  //mode before or after
                  IF (sv_CoreData[i].iCoreInPriority = sv_CoreData[k].iCoreInPriority) THEN
                     //same priority -> alarm
                     bSetAlarm := TRUE;
                  END_IF;
               END_IF;

               IF bSetAlarm THEN
                  //same mode and same priority -> alarm
                     SET_ALARM(Name := erEqualCorePriority,
                               SubID1 := i,
                               SubID2 := cMoveIn,
                               SubID3 := k,
                               SubID4 := cMoveIn);
               END_IF;
            END_IF; //end_if core in priority

            //compare core out priority with core out priority of all other cores
            IF (sv_CoreData[i].OutMode = sv_CoreData[k].OutMode) THEN
               //same mode -> check priority

               bSetAlarm := FALSE;
               IF (sv_CoreData[i].OutMode = nDuringMoldOpen) THEN
                  //mode "during" -> also consider sv_bCoresParallelToMold and the according position
                  IF sv_bCoresParallelToMold THEN
                     IF (sv_CoreData[i].iCoreOutPriority = sv_CoreData[k].iCoreOutPriority) THEN
                        //cores parallel to mold and same priority -> alarm
                        bSetAlarm := TRUE;
                     END_IF;
                  ELSE
                     IF (sv_CoreData[i].rCoreOutPosition = sv_CoreData[k].rCoreOutPosition) AND
                        (sv_CoreData[i].iCoreOutPriority = sv_CoreData[k].iCoreOutPriority) THEN
                        //cores not parallel and priority and position equal -> alarm
                        bSetAlarm := TRUE;
                     END_IF;
                  END_IF;
               ELSE
                  //mode before or after
                  IF (sv_CoreData[i].iCoreOutPriority = sv_CoreData[k].iCoreOutPriority) THEN
                     //same priority -> alarm
                     bSetAlarm := TRUE;
                  END_IF;
               END_IF;

               IF bSetAlarm THEN
                  //same mode and same priority -> alarm
                     SET_ALARM(Name := erEqualCorePriority,
                               SubID1 := i,
                               SubID2 := cMoveOut,
                               SubID3 := k,
                               SubID4 := cMoveOut);
               END_IF;
            END_IF; //end_if core out priority

         END_IF; //end_if core k
      END_FOR;  //end_for core k
   END_IF; //end_if core i available and activated
END_FOR;

STOP_PROCESS_ALGORITHM();

@END_Body

@@@BEG_Comment@@@
@TL(0)

@@@END_Comment@@@

@BEG_Body
@TL(18)
(**************************************** WARNING ********************************************
 *** The KEBA Kemro K2 System including software is not intended for safety control tasks! ***
 ***                       For further information see Comment tab!                        ***
 *********************************************************************************************)

//correct init value of core out priority (-1)
FOR i := 1 TO cMaxDeviceIndex DO
   IF sv_CoreData[i].bAvailable AND sv_CoreData[i].iCoreOutPriority = -1 THEN
      IF i = 1 THEN
         //first core gets highest number (= number of available cores)
         sv_CoreData[i].iCoreOutPriority := sv_NumberOfDevices[cCompCore];
      ELSE
         //other cores get lower number than the predecessor
         sv_CoreData[i].iCoreOutPriority := sv_CoreData[(i - 1)].iCoreOutPriority - 1;
      END_IF;
   END_IF;
END_FOR;

@END_Body

@@@BEG_Comment@@@
@TL(0)

@@@END_Comment@@@
@END_Body

@END_Contents
@@@BEG_Password@@@
M2hzZmhrMw==
@@@END_Password@@@

(* ---- ABIoForceState.pu ---- *)
IMPORT_OVER_LISTFILE
 SET_ALARM
, KCAT_GetHandle
, KCAT_GetIoState_Data
, KCAT_HandleData
, KCAT_Status
, KSYS_Status

END_IMPORT

ALGORITHM_BLOCK ABIoForceState #DUMMY_EDIT_BLOCK

SYSTEM_OBJECT
 TaskSlow : TASK;
 erAnyIoForced : ALARM;
END_OBJECT

PROCESS_ALGORITHM paCheckIoForceState ON TaskSlow AUTOSTART

VAR
 bIoForced : BOOL (* SET_ALARM called *);
 bInit : BOOL;
 iRed : DINT (* measurement reduction *);
 pbExhibitionMode : REFTO BOOL;
 IoStateDataOnboard : KCAT_GetIoState_Data;
 HandleDataOnboard : KCAT_HandleData;
 Status : KCAT_Status;
 Status2 : KSYS_Status;
END_VAR
#BEGIN_EDIT_BLOCK
(**************************************** WARNING ********************************************
 *** The KEBA Kemro K2 System including software is not intended for safety control tasks! ***
 ***                       For further information see Comment tab!                        ***
 *********************************************************************************************)

IF NOT bInit THEN
   HandleDataOnboard := KCAT_GetHandle(Name := 'IO.ONBOARD');
   pbExhibitionMode := GET_SYNC_REFTO('simulation.sv_bExhibitionMode', T#0s, Status2);
   bInit := TRUE;
END_IF;

IF ((Status2 = KSYS_Status_OK) AND pbExhibitionMode^) THEN
   // do not show erAnyIoForced alarm in exhibition mode
   IF bIoForced THEN
      RESET_ALARM(Name := erAnyIoForced);
      bIoForced := FALSE;
   END_IF;
   RETURN;
END_IF;

// measurement reduction factor
IF iRed = 0 THEN
   iRed := 5;
ELSE
   iRed := iRed - 1;
   RETURN;
END_IF;

IF (HandleDataOnboard.Status = KCAT_Status_OK) THEN
   Status := KCAT_GetIoState(Handle := HandleDataOnboard.Handle, State := IoStateDataOnboard);

   IF (IoStateDataOnboard.IoStateBits.ForcedSubTree AND NOT bIoForced) THEN
      SET_ALARM(Name := erAnyIoForced);
      bIoForced := TRUE;

   ELSIF (NOT IoStateDataOnboard.IoStateBits.ForcedSubTree AND bIoForced) THEN
      RESET_ALARM(Name := erAnyIoForced);
      bIoForced := FALSE;
   END_IF;
END_IF;

;#END_EDIT_BLOCK END_ALGORITHM

END_ALGORITHM_BLOCK

#END_OF_IEC_PART

@Puma @IecEditor 6 97 @Pou 25
@@@BEG_Comment@@@

@@@END_Comment@@@

@BEG_Contents

@BEG_Func
@RT(17)FuncTreeContainer
2
@Var @RT(9)SET_ALARM @RT(0) @T @T @DERIVED 0 @F @RT(23)KEBA_STANDARD_PROCEDURE @F
@T
@BEG_Attrib
0 @RT(0) @RT(0)
@END_Attrib
1 1 @F @F @F @F

@Var @RT(14)KCAT_GetHandle @RT(0) @T @T @DERIVED 0 @F @RT(22)KEBA_STANDARD_FUNCTION @F
@T
@BEG_Attrib
0 @RT(0) @RT(0)
@END_Attrib
1 1 @F @F @F @F

@END_Func

@BEG_Const
@RT(18)ConstTreeContainer
0
@END_Const

@BEG_Export

@BEG_Kind
@ALGORITHM_BLOCK @RT(14)ABIoForceState @STRUCTURED_TEXT
@RT(0) @RT(0) @RT(0)
@END_Kind

@BEG_Dcl
@RT(16)DclTreeContainer
2
@Var @RT(8)TaskSlow @RT(0) @T @F @DT @RT(4)TASK @RT(0) @T @T @BASIC 0 @F
@F @F
@T
@BEG_Attrib
3 @RT(0) @RT(0) @RT(0)
@END_Attrib
1 7 @F @F @F @F

@Var @RT(13)erAnyIoForced @RT(0) @T @F @DT @RT(5)ALARM @RT(0) @T @T @BASIC 0 @F
@F @F
@T
@BEG_Attrib
3 @RT(0) @RT(0) @RT(0)
@END_Attrib
1 7 @F @F @F @F

@END_Dcl

@END_Export

@BEG_Body

1

@BEG_Export

@BEG_Algo
@PROCESS_ALGORITHM @RT(19)paCheckIoForceState @STRUCTURED_TEXT
@RT(0) @RT(0) @RT(8)TaskSlow @T @F
@END_Algo

@BEG_Dcl
@RT(16)DclTreeContainer
8
@Var @RT(9)bIoForced @RT(0) @T @F @DT @RT(4)BOOL @RT(0) @T @T @BASIC 0 @F
@F @F
@T
@BEG_Attrib
3 @RT(0) @RT(16)SET_ALARM called @RT(0)
@END_Attrib
1 0 @F @F @F @F

@Var @RT(5)bInit @RT(0) @T @F @DT @RT(4)BOOL @RT(0) @T @T @BASIC 0 @F
@F @F
@T
@BEG_Attrib
3 @RT(0) @RT(0) @RT(0)
@END_Attrib
1 0 @F @F @F @F

@Var @RT(4)iRed @RT(0) @T @F @DT @RT(4)DINT @RT(0) @T @T @BASIC 0 @F
@F @F
@T
@BEG_Attrib
3 @RT(0) @RT(21)measurement reduction @RT(0)
@END_Attrib
1 0 @F @F @F @F

@Var @RT(16)pbExhibitionMode @RT(0) @T @T @REFTO 0 @T @DT @RT(4)BOOL @RT(0) @T @T @BASIC 0 @F
@F @F
@T
@BEG_Attrib
3 @RT(0) @RT(0) @RT(0)
@END_Attrib
1 0 @F @F @F @F

@Var @RT(18)IoStateDataOnboard @RT(0) @T @T @DERIVED 0 @T @T @DT @RT(20)KCAT_GetIoState_Data @RT(0) @T @T @UNKNOWN 0 @F
@F @F
@T
@BEG_Attrib
3 @RT(0) @RT(0) @RT(0)
@END_Attrib
1 0 @F @F @F @F

@Var @RT(17)HandleDataOnboard @RT(0) @T @T @DERIVED 0 @T @T @DT @RT(15)KCAT_HandleData @RT(0) @T @T @UNKNOWN 0 @F
@F @F
@T
@BEG_Attrib
3 @RT(0) @RT(0) @RT(0)
@END_Attrib
1 0 @F @F @F @F

@Var @RT(6)Status @RT(0) @T @T @DERIVED 0 @T @T @DT @RT(11)KCAT_Status @RT(0) @T @T @UNKNOWN 0 @F
@F @F
@T
@BEG_Attrib
3 @RT(0) @RT(0) @RT(0)
@END_Attrib
1 0 @F @F @F @F

@Var @RT(7)Status2 @RT(0) @T @T @DERIVED 0 @T @T @DT @RT(11)KSYS_Status @RT(0) @T @T @UNKNOWN 0 @F
@F @F
@T
@BEG_Attrib
3 @RT(0) @RT(0) @RT(0)
@END_Attrib
1 0 @F @F @F @F

@END_Dcl

@END_Export

@BEG_Body
@TL(41)
(**************************************** WARNING ********************************************
 *** The KEBA Kemro K2 System including software is not intended for safety control tasks! ***
 ***                       For further information see Comment tab!                        ***
 *********************************************************************************************)

IF NOT bInit THEN
   HandleDataOnboard := KCAT_GetHandle(Name := 'IO.ONBOARD');
   pbExhibitionMode := GET_SYNC_REFTO('simulation.sv_bExhibitionMode', T#0s, Status2);
   bInit := TRUE;
END_IF;

IF ((Status2 = KSYS_Status_OK) AND pbExhibitionMode^) THEN
   // do not show erAnyIoForced alarm in exhibition mode
   IF bIoForced THEN
      RESET_ALARM(Name := erAnyIoForced);
      bIoForced := FALSE;
   END_IF;
   RETURN;
END_IF;

// measurement reduction factor
IF iRed = 0 THEN
   iRed := 5;
ELSE
   iRed := iRed - 1;
   RETURN;
END_IF;

IF (HandleDataOnboard.Status = KCAT_Status_OK) THEN
   Status := KCAT_GetIoState(Handle := HandleDataOnboard.Handle, State := IoStateDataOnboard);

   IF (IoStateDataOnboard.IoStateBits.ForcedSubTree AND NOT bIoForced) THEN
      SET_ALARM(Name := erAnyIoForced);
      bIoForced := TRUE;

   ELSIF (NOT IoStateDataOnboard.IoStateBits.ForcedSubTree AND bIoForced) THEN
      RESET_ALARM(Name := erAnyIoForced);
      bIoForced := FALSE;
   END_IF;
END_IF;

@END_Body

@@@BEG_Comment@@@
@TL(0)

@@@END_Comment@@@
@END_Body

@END_Contents

(* ---- ABMovementRegistration.pu ---- *)
(*
This AB collects the Movement-Registration-Events which are sent by every Movement-Block.
The registrationdata is listed in 2 arrays.

@i  The movement-registration is split into 2 parts:
@i  1.The registration-event has to be sent with the
@i    registration-mode "enMoveRegModeArm".the rest of the event-data
@i    needn't be valid in this case.The event should be sent immediately after the Device-Registration
@i    is completed (sv_bInitStart -> TRUE).
@i  2.After a delaytime the registration-event has to be sent with the mode "enMoveRegModeFire",
@i    now all the eventdata have to be valid.
@i  This is necessary to make sure that no registration-events are lost, and to be able to detect the end
@i  end of the registration.
@i  When the end of the registration is detected the sv_bMoveRegisterDone flag is set TRUE.
*)

IMPORT_OVER_LISTFILE
 SET_ALARM
, ASSERT
, cMaxMoveDevicesRegistered
, cMaxMoveRegistered
, tsTraceLevel
, tyMovementRegisterList
, tDeviceMovementList
, tevMovementRegister
, tevMovementRegisterData
, ABRegisterDelay

END_IMPORT

ALGORITHM_BLOCK ABMovementRegistration #DUMMY_EDIT_BLOCK

SYSTEM_VAR
 sv_TraceLevel : tsTraceLevel;
 sv_MovementsAvailable : tyMovementRegisterList;
 sv_iMovementsAvailable : DINT;
 sv_DeviceMovements : tDeviceMovementList;
 sv_bInitDone : BOOL;
 sv_bInitStart : BOOL;
 sv_bMoveRegisterDone : BOOL;
END_VAR

SYSTEM_OBJECT
 EV_Task_3 : TASK;
 evMovementRegister : tevMovementRegister;
 erMaxMovementsExeeded : ALARM;
 erMovementRegistrationTimeout : ALARM;
 erMaxMoveRegisteredExeeded : ALARM;
 TaskMid : TASK;
 erAssert : ALARM;
 erMaxMoveDevicesExceeded : ALARM;
END_OBJECT

VAR
 miMoveRegistered : DINT;
 miMovementsToRegister : DINT;
END_VAR

EVENT_ALGORITHM evaMovementRegister ON EV_Task_3 WITH evMovementRegister

VAR_INPUT
 evMovementRegisterData : tevMovementRegisterData;
END_VAR

VAR_TEMP
 i : DINT;
END_VAR

VAR
 iRegisteredDevices : DINT;
 abRegisterDelay : ABRegisterDelay;
 dummy : DINT;
 bError : BOOL;
 b : BOOL;
 bFire : BOOL := FALSE;
END_VAR
#BEGIN_EDIT_BLOCK
(**************************************** WARNING ********************************************
 *** The KEBA Kemro K2 System including software is not intended for safety control tasks! ***
 ***                       For further information see Comment tab!                        ***
 *********************************************************************************************)

IF NOT sv_bInitDone AND NOT bError THEN

    IF evMovementRegisterData.Mode = nMoveRegModeArm THEN

        IF bFire THEN
            // arm event sent after fire events started. must never happen.
            dummy := Print('MovementRegEvent register failed, ARM %d/%d event recieved after fire event', evMovementRegisterData.DeviceId.CompId, evMovementRegisterData.DeviceId.IndexId);
        END_IF;
        b := ASSERT(NOT bFire, erAssert);

        IF sv_TraceLevel.bRegistration THEN
                dummy := Print("MovementRegEvent received: ARM %d/%d",evMovementRegisterData.DeviceId.CompId, evMovementRegisterData.DeviceId.IndexId);
        END_IF;

        //count how many movements are going to be registered
        //to be able to detect the end of the registration
        miMovementsToRegister := miMovementsToRegister + 1;

    ELSIF evMovementRegisterData.Mode = nMoveRegModeFire THEN
       bFire := TRUE;
       IF sv_TraceLevel.bRegistration THEN
            dummy := Print("MovementRegEvent received: FIRE %d/%d: %d",evMovementRegisterData.DeviceId.CompId, evMovementRegisterData.DeviceId.IndexId,evMovementRegisterData.pMovementData^.MoveId);
       END_IF;

        IF miMoveRegistered < cMaxMoveRegistered THEN

            miMoveRegistered := miMoveRegistered + 1;
            sv_iMovementsAvailable := sv_iMovementsAvailable +1;

            sv_MovementsAvailable[miMoveRegistered].DeviceId :=         evMovementRegisterData.DeviceId;
            sv_MovementsAvailable[miMoveRegistered].pbDeviceReady :=    evMovementRegisterData.pbDeviceReady;
            sv_MovementsAvailable[miMoveRegistered].pMovementData :=    evMovementRegisterData.pMovementData;

            FOR i := 1 TO cMaxMoveDevicesRegistered DO

                IF sv_DeviceMovements[i].DeviceId = evMovementRegisterData.DeviceId OR (i > iRegisteredDevices) THEN

                    IF i > iRegisteredDevices THEN
                         iRegisteredDevices := iRegisteredDevices + 1;
                    END_IF;

                    //add DeviceInfos
                    sv_DeviceMovements[i].DeviceId := evMovementRegisterData.DeviceId;
                    sv_DeviceMovements[i].pbDeviceReady := evMovementRegisterData.pbDeviceReady;
                    //add MovementData
                    IF sv_DeviceMovements[i].iNumberOfMovements < cMaxDeviceMovements THEN
                        sv_DeviceMovements[i].iNumberOfMovements := sv_DeviceMovements[i].iNumberOfMovements + 1;
                        sv_DeviceMovements[i].Movements[sv_DeviceMovements[i].iNumberOfMovements] := evMovementRegisterData.pMovementData;
                    ELSE
                        bError := TRUE;
                        // too much movements per device registered
                        SET_ALARM(Name := erMaxMovementsExeeded,
                                SubID1 := evMovementRegisterData.DeviceId.CompId,
                                SubID2 := evMovementRegisterData.DeviceId.IndexId,
                                SubID3 := cMaxDeviceMovements);
                    END_IF;
                    EXIT;
                ELSIF (iRegisteredDevices = cMaxMoveDevicesRegistered) THEN
                    //too much devices that contain movements
                    bError := TRUE;
                    SET_ALARM(Name := erMaxMoveDevicesExceeded,
                              SubID1 := cMaxMoveDevicesRegistered);
                    EXIT;
                END_IF;

            END_FOR;

            IF miMoveRegistered = miMovementsToRegister THEN
                // registration finished
                sv_bMoveRegisterDone := TRUE;
                //reset delaytime generator
                abRegisterDelay.aReset();
            END_IF;
        ELSE
            // cMaxMoveRegistered exeeded
            bError := TRUE;
            SET_ALARM(Name := erMaxMoveRegisteredExeeded,
                    SubID1 := cMaxMoveRegistered);
        END_IF;
    END_IF;
END_IF;

;#END_EDIT_BLOCK END_ALGORITHM

PROCESS_ALGORITHM paRegistrationTimeOut ON TaskMid AUTOSTART

VAR
 MoveRegisteredOld : DINT;
 dummy : DINT;
END_VAR

(* IecGraph-Code *)

(* init step *)
INITIAL_STEP Step1:
END_STEP

(* steps *)
STEP TIMEOUT:
Action2 (P);
END_STEP

ACTION Action2: #BEGIN_EDIT_BLOCK
MoveRegisteredOld := miMoveRegistered

;#END_EDIT_BLOCK END_ACTION (*Action2*)
STEP ERROR:
Action6 (P);
END_STEP

ACTION Action6: #BEGIN_EDIT_BLOCK
SET_ALARM(Name := erMovementRegistrationTimeout);
dummy := Print("Timeout during movement registration: %i of %i movements registered",miMoveRegistered,miMovementsToRegister);

;#END_EDIT_BLOCK END_ACTION (*Action6*)
STEP END:
Action3 (P);
END_STEP

ACTION Action3: #BEGIN_EDIT_BLOCK
STOP_PROCESS_ALGORITHM();

;#END_EDIT_BLOCK END_ACTION (*Action3*)

(* transitions *)
TRANSITION Trans1 (* Trans1 *) FROM Step1 TO TIMEOUT :=  #BEGIN_EDIT_BLOCK
sv_bInitStart
;#END_EDIT_BLOCK
END_TRANSITION

TRANSITION Trans2 (* Trans2 *) FROM TIMEOUT TO ERROR :=  #BEGIN_EDIT_BLOCK
TIMEOUT.T > T#10s
;#END_EDIT_BLOCK
END_TRANSITION

TRANSITION Trans3 (* Trans3 *) FROM TIMEOUT TO TIMEOUT :=  #BEGIN_EDIT_BLOCK
miMoveRegistered
> MoveRegisteredOld
;#END_EDIT_BLOCK
END_TRANSITION

TRANSITION Trans6 (* Trans6 *) FROM TIMEOUT TO END :=  #BEGIN_EDIT_BLOCK
sv_bInitDone
;#END_EDIT_BLOCK
END_TRANSITION

GO_ON_TRANSITION Trans7 (* Trans7 *) FROM ERROR TO END :=  #BEGIN_EDIT_BLOCK
TRUE
;#END_EDIT_BLOCK
END_TRANSITION

(* end IecGraph-Code *)
(* sfc-code *)
(* end sfc-code *)

END_ALGORITHM

END_ALGORITHM_BLOCK

#END_OF_IEC_PART

@Puma @IecEditor 6 96 @Pou 25
@@@BEG_Comment@@@
This AB collects the Movement-Registration-Events which are sent by every Movement-Block.
The registrationdata is listed in 2 arrays.

@i  The movement-registration is split into 2 parts:
@i  1.The registration-event has to be sent with the
@i    registration-mode "enMoveRegModeArm".the rest of the event-data
@i    needn't be valid in this case.The event should be sent immediately after the Device-Registration
@i    is completed (sv_bInitStart -> TRUE).
@i  2.After a delaytime the registration-event has to be sent with the mode "enMoveRegModeFire",
@i    now all the eventdata have to be valid.
@i  This is necessary to make sure that no registration-events are lost, and to be able to detect the end
@i  end of the registration.
@i  When the end of the registration is detected the sv_bMoveRegisterDone flag is set TRUE.
@@@END_Comment@@@

@BEG_Contents

@BEG_Func
@RT(17)FuncTreeContainer
2
@Var @RT(9)SET_ALARM @RT(0) @T @T @DERIVED 0 @F @RT(23)KEBA_STANDARD_PROCEDURE @F
@T
@BEG_Attrib
0 @RT(0) @RT(0)
@END_Attrib
1 1 @F @F @F @F

@Var @RT(6)ASSERT @RT(0) @T @T @DERIVED 0 @F @RT(8)FUNCTION @F
@T
@BEG_Attrib
0 @RT(0) @RT(0)
@END_Attrib
1 1 @F @F @F @F

@END_Func

@BEG_Const
@RT(18)ConstTreeContainer
2
@Var @RT(25)cMaxMoveDevicesRegistered @RT(0) @T @F @DT @RT(4)DINT @RT(0) @T @T @BASIC 0 @F
@F @F
@T
@BEG_Attrib
0 @RT(2)10 @RT(49)max number of devices which are serving movements
@END_Attrib
1 1 @F @F @F @F

@Var @RT(18)cMaxMoveRegistered @RT(0) @T @F @DT @RT(4)DINT @RT(0) @T @T @BASIC 0 @F
@F @F
@T
@BEG_Attrib
0 @RT(3)150 @RT(38)maximum number of registered movements
@END_Attrib
1 1 @F @F @F @F

@END_Const

@BEG_Export

@BEG_Kind
@ALGORITHM_BLOCK @RT(22)ABMovementRegistration @STRUCTURED_TEXT
@RT(0) @RT(0) @RT(0)
@END_Kind

@BEG_Dcl
@RT(16)DclTreeContainer
17
@Var @RT(9)EV_Task_3 @RT(0) @T @T @RENAMED 0 @T @T @DT @RT(4)TASK @RT(0) @T @T @BASIC 0 @F
@F @F
@T
@BEG_Attrib
3 @RT(0) @RT(0) @RT(0)
@END_Attrib
1 7 @F @F @F @F

@Var @RT(13)sv_TraceLevel @RT(0) @T @T @DERIVED 0 @T @T @DT @RT(12)tsTraceLevel @RT(0) @T @T @UNKNOWN 0 @F
@F @F
@T
@BEG_Attrib
3 @RT(0) @RT(0) @RT(0)
@END_Attrib
1 8 @F @F @F @F

@Var @RT(21)sv_MovementsAvailable @RT(0) @T @T @DERIVED 0 @T @T @DT @RT(22)tyMovementRegisterList @RT(0) @T @T @UNKNOWN 0 @F
@F @F
@T
@BEG_Attrib
3 @RT(0) @RT(0) @RT(0)
@END_Attrib
1 8 @F @F @F @F

@Var @RT(22)sv_iMovementsAvailable @RT(0) @T @F @DT @RT(4)DINT @RT(0) @T @T @BASIC 0 @F
@F @F
@T
@BEG_Attrib
3 @RT(0) @RT(0) @RT(0)
@END_Attrib
1 8 @F @F @F @F

@Var @RT(18)sv_DeviceMovements @RT(0) @T @T @DERIVED 0 @T @T @DT @RT(19)tDeviceMovementList @RT(0) @T @T @UNKNOWN 0 @F
@F @F
@T
@BEG_Attrib
3 @RT(0) @RT(0) @RT(0)
@END_Attrib
1 8 @F @F @F @F

@Var @RT(18)evMovementRegister @RT(0) @T @T @RENAMED 0 @T @T @DT @RT(19)tevMovementRegister @RT(0) @T @T @UNKNOWN 0 @F
@F @F
@T
@BEG_Attrib
3 @RT(0) @RT(0) @RT(0)
@END_Attrib
1 7 @F @F @F @F

@Var @RT(21)erMaxMovementsExeeded @RT(0) @T @F @DT @RT(5)ALARM @RT(0) @T @T @BASIC 0 @F
@F @F
@T
@BEG_Attrib
3 @RT(0) @RT(0) @RT(0)
@END_Attrib
1 7 @F @F @F @F

@Var @RT(29)erMovementRegistrationTimeout @RT(0) @T @F @DT @RT(5)ALARM @RT(0) @T @T @BASIC 0 @F
@F @F
@T
@BEG_Attrib
3 @RT(0) @RT(0) @RT(0)
@END_Attrib
1 7 @F @F @F @F

@Var @RT(26)erMaxMoveRegisteredExeeded @RT(0) @T @F @DT @RT(5)ALARM @RT(0) @T @T @BASIC 0 @F
@F @F
@T
@BEG_Attrib
3 @RT(0) @RT(0) @RT(0)
@END_Attrib
1 7 @F @F @F @F

@Var @RT(12)sv_bInitDone @RT(0) @T @F @DT @RT(4)BOOL @RT(0) @T @T @BASIC 0 @F
@F @F
@T
@BEG_Attrib
3 @RT(0) @RT(0) @RT(0)
@END_Attrib
1 8 @F @F @F @F

@Var @RT(13)sv_bInitStart @RT(0) @T @F @DT @RT(4)BOOL @RT(0) @T @T @BASIC 0 @F
@F @F
@T
@BEG_Attrib
3 @RT(0) @RT(0) @RT(0)
@END_Attrib
1 8 @F @F @F @F

@Var @RT(16)miMoveRegistered @RT(0) @T @F @DT @RT(4)DINT @RT(0) @T @T @BASIC 0 @F
@F @F
@T
@BEG_Attrib
3 @RT(0) @RT(0) @RT(0)
@END_Attrib
1 0 @F @F @F @F

@Var @RT(21)miMovementsToRegister @RT(0) @T @F @DT @RT(4)DINT @RT(0) @T @T @BASIC 0 @F
@F @F
@T
@BEG_Attrib
3 @RT(0) @RT(0) @RT(0)
@END_Attrib
1 0 @F @F @F @F

@Var @RT(7)TaskMid @RT(0) @T @T @RENAMED 0 @T @T @DT @RT(4)TASK @RT(0) @T @T @BASIC 0 @F
@F @F
@T
@BEG_Attrib
3 @RT(0) @RT(0) @RT(0)
@END_Attrib
1 7 @F @F @F @F

@Var @RT(20)sv_bMoveRegisterDone @RT(0) @T @F @DT @RT(4)BOOL @RT(0) @T @T @BASIC 0 @F
@F @F
@T
@BEG_Attrib
3 @RT(0) @RT(0) @RT(0)
@END_Attrib
1 8 @F @F @F @F

@Var @RT(8)erAssert @RT(0) @T @F @DT @RT(5)ALARM @RT(0) @T @T @BASIC 0 @F
@F @F
@T
@BEG_Attrib
3 @RT(0) @RT(0) @RT(0)
@END_Attrib
1 7 @F @F @F @F

@Var @RT(24)erMaxMoveDevicesExceeded @RT(0) @T @F @DT @RT(5)ALARM @RT(0) @T @T @BASIC 0 @F
@F @F
@T
@BEG_Attrib
3 @RT(0) @RT(0) @RT(0)
@END_Attrib
1 7 @F @F @F @F

@END_Dcl

@END_Export

@BEG_Body

2

@BEG_Export

@BEG_Algo
@EVENT_ALGORITHM @RT(19)evaMovementRegister @STRUCTURED_TEXT
@RT(0) @RT(18)evMovementRegister @RT(9)EV_Task_3 @F @F
@END_Algo

@BEG_Dcl
@RT(16)DclTreeContainer
8
@Var @RT(22)evMovementRegisterData @RT(0) @T @T @DERIVED 0 @T @T @DT @RT(23)tevMovementRegisterData @RT(0) @T @T @UNKNOWN 0 @F
@F @F
@T
@BEG_Attrib
3 @RT(0) @RT(0) @RT(0)
@END_Attrib
1 1 @F @F @F @F

@Var @RT(1)i @RT(0) @T @F @DT @RT(4)DINT @RT(0) @T @T @BASIC 0 @F
@F @F
@T
@BEG_Attrib
3 @RT(0) @RT(0) @RT(0)
@END_Attrib
1 4 @F @F @F @F

@Var @RT(18)iRegisteredDevices @RT(0) @T @F @DT @RT(4)DINT @RT(0) @T @T @BASIC 0 @F
@F @F
@T
@BEG_Attrib
3 @RT(0) @RT(0) @RT(0)
@END_Attrib
1 0 @F @F @F @F

@Var @RT(15)abRegisterDelay @RT(0) @T @T @DERIVED 0 @T @T @DT @RT(15)ABRegisterDelay @RT(0) @T @T @UNKNOWN 0 @F
@F @F
@T
@BEG_Attrib
3 @RT(0) @RT(0) @RT(0)
@END_Attrib
1 0 @F @F @F @F

@Var @RT(5)dummy @RT(0) @T @F @DT @RT(4)DINT @RT(0) @T @T @BASIC 0 @F
@F @F
@T
@BEG_Attrib
3 @RT(0) @RT(0) @RT(0)
@END_Attrib
1 0 @F @F @F @F

@Var @RT(6)bError @RT(0) @T @F @DT @RT(4)BOOL @RT(0) @T @T @BASIC 0 @F
@F @F
@T
@BEG_Attrib
3 @RT(0) @RT(0) @RT(0)
@END_Attrib
1 0 @F @F @F @F

@Var @RT(1)b @RT(0) @T @F @DT @RT(4)BOOL @RT(0) @T @T @BASIC 0 @F
@F @F
@T
@BEG_Attrib
3 @RT(0) @RT(0) @RT(0)
@END_Attrib
1 0 @F @F @F @F

@Var @RT(5)bFire @RT(0) @T @F @DT @RT(4)BOOL @RT(0) @T @T @BASIC 0 @F
@F @F
@T
@BEG_Attrib
3 @RT(5)FALSE @RT(0) @RT(0)
@END_Attrib
1 0 @F @F @F @F

@END_Dcl

@END_Export

@BEG_Export

@BEG_Algo
@PROCESS_ALGORITHM @RT(21)paRegistrationTimeOut @SEQUENTIAL_FLOW_CHART
@RT(0) @RT(0) @RT(7)TaskMid @T @F
@END_Algo

@BEG_Dcl
@RT(16)DclTreeContainer
2
@Var @RT(17)MoveRegisteredOld @RT(0) @T @F @DT @RT(4)DINT @RT(0) @T @T @BASIC 0 @F
@F @F
@T
@BEG_Attrib
3 @RT(0) @RT(0) @RT(0)
@END_Attrib
1 0 @F @F @F @F

@Var @RT(5)dummy @RT(0) @T @F @DT @RT(4)DINT @RT(0) @T @T @BASIC 0 @F
@F @F
@T
@BEG_Attrib
3 @RT(0) @RT(0) @RT(0)
@END_Attrib
1 0 @F @F @F @F

@END_Dcl

@END_Export

@BEG_Body
@TL(87)
(**************************************** WARNING ********************************************
 *** The KEBA Kemro K2 System including software is not intended for safety control tasks! ***
 ***                       For further information see Comment tab!                        ***
 *********************************************************************************************)

IF NOT sv_bInitDone AND NOT bError THEN

    IF evMovementRegisterData.Mode = nMoveRegModeArm THEN

        IF bFire THEN
            // arm event sent after fire events started. must never happen.
            dummy := Print('MovementRegEvent register failed, ARM %d/%d event recieved after fire event', evMovementRegisterData.DeviceId.CompId, evMovementRegisterData.DeviceId.IndexId);
        END_IF;
        b := ASSERT(NOT bFire, erAssert);

        IF sv_TraceLevel.bRegistration THEN
                dummy := Print("MovementRegEvent received: ARM %d/%d",evMovementRegisterData.DeviceId.CompId, evMovementRegisterData.DeviceId.IndexId);
        END_IF;

        //count how many movements are going to be registered
        //to be able to detect the end of the registration
        miMovementsToRegister := miMovementsToRegister + 1;

    ELSIF evMovementRegisterData.Mode = nMoveRegModeFire THEN
       bFire := TRUE;
       IF sv_TraceLevel.bRegistration THEN
            dummy := Print("MovementRegEvent received: FIRE %d/%d: %d",evMovementRegisterData.DeviceId.CompId, evMovementRegisterData.DeviceId.IndexId,evMovementRegisterData.pMovementData^.MoveId);
       END_IF;

        IF miMoveRegistered < cMaxMoveRegistered THEN

            miMoveRegistered := miMoveRegistered + 1;
            sv_iMovementsAvailable := sv_iMovementsAvailable +1;

            sv_MovementsAvailable[miMoveRegistered].DeviceId :=         evMovementRegisterData.DeviceId;
            sv_MovementsAvailable[miMoveRegistered].pbDeviceReady :=    evMovementRegisterData.pbDeviceReady;
            sv_MovementsAvailable[miMoveRegistered].pMovementData :=    evMovementRegisterData.pMovementData;

            FOR i := 1 TO cMaxMoveDevicesRegistered DO

                IF sv_DeviceMovements[i].DeviceId = evMovementRegisterData.DeviceId OR (i > iRegisteredDevices) THEN

                    IF i > iRegisteredDevices THEN
                         iRegisteredDevices := iRegisteredDevices + 1;
                    END_IF;

                    //add DeviceInfos
                    sv_DeviceMovements[i].DeviceId := evMovementRegisterData.DeviceId;
                    sv_DeviceMovements[i].pbDeviceReady := evMovementRegisterData.pbDeviceReady;
                    //add MovementData
                    IF sv_DeviceMovements[i].iNumberOfMovements < cMaxDeviceMovements THEN
                        sv_DeviceMovements[i].iNumberOfMovements := sv_DeviceMovements[i].iNumberOfMovements + 1;
                        sv_DeviceMovements[i].Movements[sv_DeviceMovements[i].iNumberOfMovements] := evMovementRegisterData.pMovementData;
                    ELSE
                        bError := TRUE;
                        // too much movements per device registered
                        SET_ALARM(Name := erMaxMovementsExeeded,
                                SubID1 := evMovementRegisterData.DeviceId.CompId,
                                SubID2 := evMovementRegisterData.DeviceId.IndexId,
                                SubID3 := cMaxDeviceMovements);
                    END_IF;
                    EXIT;
                ELSIF (iRegisteredDevices = cMaxMoveDevicesRegistered) THEN
                    //too much devices that contain movements
                    bError := TRUE;
                    SET_ALARM(Name := erMaxMoveDevicesExceeded,
                              SubID1 := cMaxMoveDevicesRegistered);
                    EXIT;
                END_IF;

            END_FOR;

            IF miMoveRegistered = miMovementsToRegister THEN
                // registration finished
                sv_bMoveRegisterDone := TRUE;
                //reset delaytime generator
                abRegisterDelay.aReset();
            END_IF;
        ELSE
            // cMaxMoveRegistered exeeded
            bError := TRUE;
            SET_ALARM(Name := erMaxMoveRegisteredExeeded,
                    SubID1 := cMaxMoveRegistered);
        END_IF;
    END_IF;
END_IF;

@END_Body

@@@BEG_Comment@@@
@TL(0)

@@@END_Comment@@@

@BEG_SfcBody
7 6 8

@BEG_SfcData 2
@StepSeq @RT(4)sseq @F 7
@Step @RT(5)Step1 @F @T @F @F @RT(0) @F
@AcbCont @RT(7)unnamed @F 0

@Trans @RT(6)Trans1 @F @T @F @F @T @T @TL(2)
sv_bInitStart

@RT(6)Trans1 @F
@Step @RT(7)TIMEOUT @F @F @T @F @RT(0) @F
@AcbCont @RT(7)unnamed @F 1
@Acb @RT(7)Action2 @F @T @RT(1)P @RT(0) @F @F @T @TL(2)
MoveRegisteredOld := miMoveRegistered

@F

@AltBranch @RT(3)alt @F 3
@TransSeq @RT(4)tseq @F 1
@Trans @RT(6)Trans2 @F @T @F @F @T @T @TL(2)
TIMEOUT.T > T#10s

@RT(6)Trans2 @F

@TransSeq @RT(4)tseq @F 2
@Trans @RT(6)Trans3 @F @T @F @F @T @T @TL(3)
miMoveRegistered
> MoveRegisteredOld

@RT(6)Trans3 @F
@Goto @RT(7)TIMEOUT @F @F

@TransSeq @RT(4)tseq @F 2
@Trans @RT(6)Trans6 @F @T @F @F @T @T @TL(2)
sv_bInitDone

@RT(6)Trans6 @F
@Goto @RT(3)END @F @F

@Step @RT(5)ERROR @F @F @F @F @RT(0) @F
@AcbCont @RT(7)unnamed @F 1
@Acb @RT(7)Action6 @F @T @RT(1)P @RT(0) @F @F @T @TL(4)
SET_ALARM(Name := erMovementRegistrationTimeout);
dummy := Print("Timeout during movement registration: %i of %i movements registered",miMoveRegistered,miMovementsToRegister);

@F

@Trans @RT(6)Trans7 @F @T @F @F @T @F @TL(2)
TRUE

@RT(6)Trans7 @F
@Step @RT(3)END @F @F @T @F @RT(0) @F
@AcbCont @RT(7)unnamed @F 1
@Acb @RT(7)Action3 @F @T @RT(1)P @RT(0) @F @F @T @TL(2)
STOP_PROCESS_ALGORITHM();

@F

@END_SfcData
@SaActions 0
@SaTrans 0
@SaExits 0
@END_SfcBody

@@@BEG_Comment@@@
@TL(0)

@@@END_Comment@@@
@END_Body

@END_Contents

(* ---- FPlausCoreInMode.pu ---- *)
IMPORT_OVER_LISTFILE
 GET_SYNC_REFTO
, cOptionHydraulic
, tyCoreInModePlaus
, KSYS_Status
, tOptionId

END_IMPORT

PLAUSIBILITY_FUNCTION FPlausCoreInMode : tyCoreInModePlaus

VAR_INPUT
 DeviceClass : INT;
 Userlevel : INT;
END_VAR

VAR
 s : KSYS_Status;
 pOptions : REFTO tOptionId;
 b2Platen : BOOL;
END_VAR
#BEGIN_EDIT_BLOCK
(**************************************** WARNING ********************************************
 *** The KEBA Kemro K2 System including software is not intended for safety control tasks! ***
 ***                       For further information see Comment tab!                        ***
 *********************************************************************************************)

//selectable modes depend on machine type
//2 platen machines have some additional modes
pOptions := GET_SYNC_REFTO('Mold1.sv_Options', T#0s, s);
IF s = KSYS_Status_OK THEN
   b2Platen := (pOptions^ AND cSubOptionMold2Platen) = cSubOptionMold2Platen;
END_IF;

FPlausCoreInMode[1] := nBefMoldClose;
FPlausCoreInMode[2] := nDuringMoldClose;
FPlausCoreInMode[3] := nAfterMoldClose;

IF b2Platen THEN
   FPlausCoreInMode[4] := nAfterMoldNutsClose;
   FPlausCoreInMode[5] := nAfterHighPress;
ELSE
   FPlausCoreInMode[4] := nAfterMoldClose;
   FPlausCoreInMode[5] := nAfterMoldClose;
END_IF;

;#END_EDIT_BLOCK END_FUNCTION

#END_OF_IEC_PART

@Puma @IecEditor 6 114 @Pou 25
@@@BEG_Comment@@@

@@@END_Comment@@@

@BEG_Contents

@BEG_Func
@RT(17)FuncTreeContainer
1
@Var @RT(14)GET_SYNC_REFTO @RT(0) @T @T @DERIVED 0 @F @RT(22)KEBA_STANDARD_FUNCTION @F
@T
@BEG_Attrib
0 @RT(0) @RT(0)
@END_Attrib
1 1 @F @F @F @F

@END_Func

@BEG_Const
@RT(18)ConstTreeContainer
1
@Var @RT(16)cOptionHydraulic @RT(0) @T @F @DT @RT(5)DWORD @RT(0) @T @T @BASIC 0 @F
@F @F
@T
@BEG_Attrib
0 @RT(5)16#01 @RT(26)Hydraulic device, LSB is 1
@END_Attrib
1 1 @F @F @F @F

@END_Const

@BEG_Export

@BEG_Kind
@PLAUSIBILITY_FUNCTION @RT(16)FPlausCoreInMode @STRUCTURED_TEXT
@RT(17)tyCoreInModePlaus @RT(0) @RT(0)
@END_Kind

@BEG_Dcl
@RT(16)DclTreeContainer
5
@Var @RT(11)DeviceClass @RT(0) @T @F @DT @RT(3)INT @RT(0) @T @T @BASIC 0 @F
@F @F
@T
@BEG_Attrib
3 @RT(0) @RT(0) @RT(0)
@END_Attrib
0 1 @F @F @F @F

@Var @RT(9)Userlevel @RT(0) @T @F @DT @RT(3)INT @RT(0) @T @T @BASIC 0 @F
@F @F
@T
@BEG_Attrib
3 @RT(0) @RT(0) @RT(0)
@END_Attrib
0 1 @F @F @F @F

@Var @RT(1)s @RT(0) @T @T @DERIVED 0 @T @T @DT @RT(11)KSYS_Status @RT(0) @T @T @UNKNOWN 0 @F
@F @F
@T
@BEG_Attrib
3 @RT(0) @RT(0) @RT(0)
@END_Attrib
1 0 @F @F @F @F

@Var @RT(8)pOptions @RT(0) @T @T @REFTO 0 @F @DERIVED 0 @T @T @DT @RT(9)tOptionId @RT(0) @T @T @UNKNOWN 0 @F
@F @F
@T
@BEG_Attrib
3 @RT(0) @RT(0) @RT(0)
@END_Attrib
1 0 @F @F @F @F

@Var @RT(8)b2Platen @RT(0) @T @F @DT @RT(4)BOOL @RT(0) @T @T @BASIC 0 @F
@F @F
@T
@BEG_Attrib
3 @RT(0) @RT(0) @RT(0)
@END_Attrib
1 0 @F @F @F @F

@END_Dcl

@END_Export

@BEG_Body
@TL(28)
(**************************************** WARNING ********************************************
 *** The KEBA Kemro K2 System including software is not intended for safety control tasks! ***
 ***                       For further information see Comment tab!                        ***
 *********************************************************************************************)

//selectable modes depend on machine type
//2 platen machines have some additional modes
pOptions := GET_SYNC_REFTO('Mold1.sv_Options', T#0s, s);
IF s = KSYS_Status_OK THEN
   b2Platen := (pOptions^ AND cSubOptionMold2Platen) = cSubOptionMold2Platen;
END_IF;

FPlausCoreInMode[1] := nBefMoldClose;
FPlausCoreInMode[2] := nDuringMoldClose;
FPlausCoreInMode[3] := nAfterMoldClose;

IF b2Platen THEN
   FPlausCoreInMode[4] := nAfterMoldNutsClose;
   FPlausCoreInMode[5] := nAfterHighPress;
ELSE
   FPlausCoreInMode[4] := nAfterMoldClose;
   FPlausCoreInMode[5] := nAfterMoldClose;
END_IF;

@END_Body

@END_Contents

(* ---- FPlausCoreOutMode.pu ---- *)
IMPORT_OVER_LISTFILE
 GET_SYNC_REFTO
, cOptionHydraulic
, tyCoreOutModePlaus
, KSYS_Status
, tOptionId

END_IMPORT

PLAUSIBILITY_FUNCTION FPlausCoreOutMode : tyCoreOutModePlaus

VAR_INPUT
 DeviceClass : INT;
 Userlevel : INT;
END_VAR

VAR
 s : KSYS_Status;
 pOptions : REFTO tOptionId;
 b2Platen : BOOL;
END_VAR
#BEGIN_EDIT_BLOCK
(**************************************** WARNING ********************************************
 *** The KEBA Kemro K2 System including software is not intended for safety control tasks! ***
 ***                       For further information see Comment tab!                        ***
 *********************************************************************************************)

//selectable modes depend on machine type
//2 platen machines have some additional modes
pOptions := GET_SYNC_REFTO('Mold1.sv_Options', T#0s, s);
IF s = KSYS_Status_OK THEN
   b2Platen := (pOptions^ AND cSubOptionMold2Platen) = cSubOptionMold2Platen;
END_IF;

FPlausCoreOutMode[1] := nBefMoldOpen;
FPlausCoreOutMode[2] := nDuringMoldOpen;
FPlausCoreOutMode[3] := nAfterMoldOpen;

IF b2Platen THEN
   FPlausCoreOutMode[4] := nBeforeHiPressRel;
   FPlausCoreOutMode[5] := nAfterHiPressRel;
   FPlausCoreOutMode[6] := nBeforeMoldNutsOpen;
ELSE
   FPlausCoreOutMode[4] := nAfterMoldOpen;
   FPlausCoreOutMode[5] := nAfterMoldOpen;
   FPlausCoreOutMode[6] := nAfterMoldOpen;
END_IF;

;#END_EDIT_BLOCK END_FUNCTION

#END_OF_IEC_PART

@Puma @IecEditor 6 114 @Pou 25
@@@BEG_Comment@@@

@@@END_Comment@@@

@BEG_Contents

@BEG_Func
@RT(17)FuncTreeContainer
1
@Var @RT(14)GET_SYNC_REFTO @RT(0) @T @T @DERIVED 0 @F @RT(22)KEBA_STANDARD_FUNCTION @F
@T
@BEG_Attrib
0 @RT(0) @RT(0)
@END_Attrib
1 1 @F @F @F @F

@END_Func

@BEG_Const
@RT(18)ConstTreeContainer
1
@Var @RT(16)cOptionHydraulic @RT(0) @T @F @DT @RT(5)DWORD @RT(0) @T @T @BASIC 0 @F
@F @F
@T
@BEG_Attrib
0 @RT(5)16#01 @RT(26)Hydraulic device, LSB is 1
@END_Attrib
1 1 @F @F @F @F

@END_Const

@BEG_Export

@BEG_Kind
@PLAUSIBILITY_FUNCTION @RT(17)FPlausCoreOutMode @STRUCTURED_TEXT
@RT(18)tyCoreOutModePlaus @RT(0) @RT(0)
@END_Kind

@BEG_Dcl
@RT(16)DclTreeContainer
5
@Var @RT(11)DeviceClass @RT(0) @T @F @DT @RT(3)INT @RT(0) @T @T @BASIC 0 @F
@F @F
@T
@BEG_Attrib
3 @RT(0) @RT(0) @RT(0)
@END_Attrib
0 1 @F @F @F @F

@Var @RT(9)Userlevel @RT(0) @T @F @DT @RT(3)INT @RT(0) @T @T @BASIC 0 @F
@F @F
@T
@BEG_Attrib
3 @RT(0) @RT(0) @RT(0)
@END_Attrib
0 1 @F @F @F @F

@Var @RT(1)s @RT(0) @T @T @DERIVED 0 @T @T @DT @RT(11)KSYS_Status @RT(0) @T @T @UNKNOWN 0 @F
@F @F
@T
@BEG_Attrib
3 @RT(0) @RT(0) @RT(0)
@END_Attrib
1 0 @F @F @F @F

@Var @RT(8)pOptions @RT(0) @T @T @REFTO 0 @F @DERIVED 0 @T @T @DT @RT(9)tOptionId @RT(0) @T @T @UNKNOWN 0 @F
@F @F
@T
@BEG_Attrib
3 @RT(0) @RT(0) @RT(0)
@END_Attrib
1 0 @F @F @F @F

@Var @RT(8)b2Platen @RT(0) @T @F @DT @RT(4)BOOL @RT(0) @T @T @BASIC 0 @F
@F @F
@T
@BEG_Attrib
3 @RT(0) @RT(0) @RT(0)
@END_Attrib
1 0 @F @F @F @F

@END_Dcl

@END_Export

@BEG_Body
@TL(30)
(**************************************** WARNING ********************************************
 *** The KEBA Kemro K2 System including software is not intended for safety control tasks! ***
 ***                       For further information see Comment tab!                        ***
 *********************************************************************************************)

//selectable modes depend on machine type
//2 platen machines have some additional modes
pOptions := GET_SYNC_REFTO('Mold1.sv_Options', T#0s, s);
IF s = KSYS_Status_OK THEN
   b2Platen := (pOptions^ AND cSubOptionMold2Platen) = cSubOptionMold2Platen;
END_IF;

FPlausCoreOutMode[1] := nBefMoldOpen;
FPlausCoreOutMode[2] := nDuringMoldOpen;
FPlausCoreOutMode[3] := nAfterMoldOpen;

IF b2Platen THEN
   FPlausCoreOutMode[4] := nBeforeHiPressRel;
   FPlausCoreOutMode[5] := nAfterHiPressRel;
   FPlausCoreOutMode[6] := nBeforeMoldNutsOpen;
ELSE
   FPlausCoreOutMode[4] := nAfterMoldOpen;
   FPlausCoreOutMode[5] := nAfterMoldOpen;
   FPlausCoreOutMode[6] := nAfterMoldOpen;
END_IF;

@END_Body

@END_Contents
